			IF mcCartesianZMoveAbsolute.Done THEN
				bMissingCaps						:= TRUE;
				bCycleDone;
				mcCartesianZMoveAbsolute.Execute	:= FALSE;
				eRunningState						:= E_CapPreScrewer.eReady;	
			END_IF
			
		ELSE
			mcCartesianZMoveAbsolute.Execute		:= NOT stParameters.bVacuumDeactivate;		
			mcCartesianZMoveAbsolute.Position		:= stParameters.lrTopZPosition;
			mcCartesianZMoveAbsolute.Acceleration	:= SEL(GVL_Recipe.iCapSorterProductType = 0 ,stParameters.lrPickerAcceleration , 150.0);//stParameters.lrPickerAcceleration;
//			mcCartesianZMoveAbsolute.Acceleration	:= stParameters.lrPickerAcceleration;
			mcCartesianZMoveAbsolute.Deceleration	:= stParameters.lrPickerAcceleration;
			mcCartesianZMoveAbsolute.Velocity		:= stParameters.lrPickerSpeed;
			tonCapCatcher.IN						:= FALSE;
			
			IF mcCartesianZMoveAbsolute.Busy OR stParameters.bVacuumDeactivate THEN
				mcCartesianZMoveAbsolute.Execute		:= FALSE;
				eRunningState 							:= E_CapPreScrewer.eTransferingVertical; 
			END_IF
			
        
		END_IF		
			
			//przepisuje do rejestrów nakretki które kartezjan pobrał
			aCapPresence[1] := bCapSucker[1];
			aCapPresence[2] := bCapSucker[2];
			aCapPresence[3] := bCapSucker[3];
			aCapPresence[4] := bCapSucker[4];						

		
		
	(*Jazda w górę, zamknięcie łapek i załączenie jazdy w bok*)	
	E_CapPreScrewer.eTransferingVertical:
		
		IF NOT bCapSucker[1] OR NOT bCapSucker[2] OR NOT bCapSucker[3] OR NOT bCapSucker[4] THEN
            bCapBlow1						:= NOT bCapSucker[1];
            bCapBlow2						:= NOT bCapSucker[2];
            bCapBlow3						:= NOT bCapSucker[3];
            bCapBlow4						:= NOT bCapSucker[4];						
			bCapsBlowON						:= TRUE;
		END_IF
		
		//Kleją się kulki 
		IF NOT stParameters.bVacuumDeactivate THEN					
			IF CartesianZAxisRef.NcToPlc.ActPos > stParameters.lrPickZPosition + 10.0 THEN
				mcCartesianZMoveAbsolute2.Execute		:= NOT stParameters.bVacuumDeactivate;		
				mcCartesianZMoveAbsolute2.Position		:= stParameters.lrTopZPosition;
				mcCartesianZMoveAbsolute2.Acceleration	:= stParameters.lrPickerAcceleration;
				mcCartesianZMoveAbsolute2.Deceleration	:= stParameters.lrPickerAcceleration;
				mcCartesianZMoveAbsolute2.Velocity		:= stParameters.lrPickerSpeed;
			END_IF
		END_IF


		IF CartesianZAxisRef.NcToPlc.ActPos > stParameters.lrCapCatcherZPosition OR (CartesianZAxisRef.NcToPlc.ActPos > stParameters.lrTopZPosition - stParameters.lrBendingDistance) THEN
			bCapCatcher1							:= TRUE;
			bCapCatcher2							:= true;
			bCapCatcher3							:= true;
			bCapCatcher4							:= true;
			tonCapCatcher.IN						:= stParameters.bVacuumDeactivate;
		END_IF	
		
		mcCartesianZMoveAbsolute.Execute		:= tonCapCatcher.Q;	
		
		//Dodać sprawdzenie czy gotowy chwytak słomek !!!!!
		//Sprawdzenie pozycji osi pionowej Z i czy wysunięty siłownik chwytaka słomek
		IF ((CartesianZAxisRef.NcToPlc.ActPos > stParameters.lrTopZPosition - stParameters.lrBendingDistance) OR
			mcCartesianZMoveAbsolute.Done) AND (tonStrawCatcherOut.Q OR NOT stParameters.bStrawCatcherON) THEN
			//Jedź osią poziomą X na pozycję pick
				mcCartesianZMoveAbsolute2.Execute		:= FALSE;
				bCapsBlowON								:= FALSE;
				eRunningState 							:= E_CapPreScrewer.eTransferingHorizontal;
				tonCapCatcher.IN						:= FALSE;
		END_IF
	
	(*Przejazd w poziomie*)	
	E_CapPreScrewer.eTransferingHorizontal:	
	
			bCapCatcher1							:= TRUE;//bCapSucker1;
			bCapCatcher2							:= TRUE;//bCapSucker2;
			bCapCatcher3							:= TRUE;//bCapSucker3;
			bCapCatcher4							:= TRUE;//bCapSucker4;
	
		mcCartesianYMoveAbsolute.Position			:= stParameters.lrPlaceYPosition;
		mcCartesianYMoveAbsolute.Acceleration		:= stParameters.lrPickerAcceleration;
		mcCartesianYMoveAbsolute.Deceleration		:= stParameters.lrPickerAcceleration;
		mcCartesianYMoveAbsolute.Velocity			:= stParameters.lrPickerSpeed;
		mcCartesianYMoveAbsolute.Execute			:= TRUE;
		
		IF (CartesianYAxisRef.NcToPlc.ActPos > 200.0 (*stParameters.lrPlaceYPosition - stParameters.lrBendingDistance*)) OR
			mcCartesianYMoveAbsolute.Done AND NOT mcCartesianZMoveAbsolute.Execute THEN			

			//Podjedź robotem w dól	
			mcCartesianZMoveAbsolute.Execute			:= TRUE;		
			mcCartesianZMoveAbsolute.Position			:= stParameters.lrCartesianCatchZPosition;
			mcCartesianZMoveAbsolute.Acceleration		:= stParameters.lrPickerAcceleration;
			mcCartesianZMoveAbsolute.Deceleration		:= stParameters.lrPickerAcceleration;
			mcCartesianZMoveAbsolute.Velocity			:= stParameters.lrPickerSpeed;
		END_IF
		
		//Jak obie pozycje osiągnięte 
		IF mcCartesianZMoveAbsolute.Done THEN
			mcCartesianZMoveAbsolute.Execute		:= FALSE;
		END_IF
			
		//Jak ak obie pozycje osiągnięte to zamykamy chwytaki i następny krok
		IF stParameters.bStrawCatcherON AND CartesianYAxisRef.NcToPlc.ActPos >= stParameters.lrPlaceYPosition THEN
			//Zamknij chwytaki słomek
			bStrawCatchersOpen						:= FALSE;
			bStrawCatchersClose						:= TRUE;	
		END_IF
		
			
		IF  mcCartesianYMoveAbsolute.Done AND mcCartesianZMoveAbsolute.Done THEN
			//Reset komendy ruchu osi
			mcCartesianYMoveAbsolute.Execute		:= FALSE;
			mcCartesianZMoveAbsolute.Execute		:= FALSE;
			
				//Ustaw pozycję wirtualnej osi tak samo jak na osi Z
			fbVirtualAxis.fPosition						:= CartesianZAxisRef.NcToPlc.ActPos;
			fbVirtualAxis.SetPosAbsClearLag(bExecute	:= TRUE);
				
				IF fbVirtualAxis.pSetPos.Busy THEN
					//Następny krok
					eRunningState						:= E_CapPreScrewer.eVerticalDownToCatchPos;	
				END_IF
		END_IF		
		
	(*Przejazd w dól do pozycji chwytanija rurki*)		
	E_CapPreScrewer.eVerticalDownToCatchPos:
		fbVirtualAxis.SetPosAbsClearLag(bExecute				:= FALSE);
		
		//Jak ak obie pozycje osiągnięte to zamykamy chwytaki i następny krok
		IF stParameters.bStrawCatcherON THEN
			//Zamknij chwytaki słomek
			bStrawCatchersOpen						:= FALSE;
			bStrawCatchersClose						:= TRUE;	
		END_IF
				
		IF tonPlacePermission.Q AND ((bCapCatcher1 OR NOT bCapCatcher1) AND (bCapCatcher2  OR NOT bCapCatcher2) AND
									(bCapCatcher3  OR NOT bCapCatcher3) AND(bCapCatcher4  OR NOT bCapCatcher4)) AND (tonStrawCatcher1Close.Q OR NOT stParameters.bStrawCatcherON) THEN				
				bCapCatcher1						:= TRUE;
				bCapCatcher2						:= TRUE;
				bCapCatcher3						:= TRUE;
				bCapCatcher4						:= TRUE;						
				eRunningState						:= E_CapPreScrewer.eAxisGearIn;
		END_IF
		
			//Następny krok
			//IF stParameters.bStrawCatcherON THEN
			//	eRunningState						:= E_CapPreScrewer.eCatching;	
			//ELSE
			//	eRunningState						:= E_CapPreScrewer.ePlacing;	
			//END_IF				
		//END_IF
	
	
	E_CapPreScrewer.eAxisGearIn:
		fbGearInCatcherAxis.Enable						:= stParameters.bStrawCatcherON;
		fbGearInCatcherAxis.GearRatio					:= 1;
		fbGearInAxisZ.Enable							:= TRUE;
		fbGearInAxisZ.GearRatio							:= SEL(stParameters.bStrawCatcherON, 1.0, 0.0000000001);
		
		
			IF (fbGearInCatcherAxis.InGear OR NOT stParameters.bStrawCatcherON) AND fbGearInAxisZ.InGear AND (tonStrawCatcher1Close.Q (*AND tonStrawCatcher2Close.Q*)
					OR (bStrawCatcherOpen1 AND bStrawCatcherOpen2 AND bStrawCatcherOpen3 AND bStrawCatcherOpen4))  THEN
				IF stParameters.bStrawCatcherON THEN
					eRunningState						:= E_CapPreScrewer.eCatching;	
				ELSE
					eRunningState						:= E_CapPreScrewer.ePlacing;	
				END_IF					
			END_IF		

	
	//Sprawdzanie czy chwytaki zamknięte i opuszczenie chwytaków do dolnej pozycji
	E_CapPreScrewer.eCatching:
		fbVirtualAxis.fPosition							:= (stParameters.LrCheckStrawCatcherActuatorZPosition - stParameters.lrStrawInsertDistance);	//Pozycja sprawdzania cofnięcia krabów
		fbVirtualAxis.fVelocity							:= SEL(stParameters.lrCatcherSpeed > 1094.0, stParameters.lrCatcherSpeed, 1094.0 );       						
		bVirtualMove									:= TRUE;				
	
	IF (CatcherAxisRef.NcToPlc.ActPos + stParameters.lrCatcherHightSV) <= (stParameters.lrCartesianCatchZPosition - (stParameters.lrCapHight + 25.0)) THEN	//+25
		fbGearInAxisZ.GearRatio								:= 1;
	END_IF
	
	//IF (CatcherAxisRef.NcToPlc.ActPos + stParameters.lrCatcherHightSV) <= (stParameters.lrCartesianCatchZPosition-(stParameters.lrCapHight)) THEN
	//	fbGearInAxisZ.GearRatio							:= 1;
	//END_IF
	
			//Otwórz chwytaki słomek
		IF CartesianZAxisRef.NcToPlc.ActPos <= stParameters.lrStrawCatcherZPosition THEN					
			bStrawCatchersOpen							:= TRUE;
			bStrawCatchersClose							:= FALSE;
			
				IF tonStrawCatcher1Open.Q AND tonStrawCatcher2Open.Q AND tonStrawCatcher3Open.Q AND tonStrawCatcher4Open.Q THEN																				
					//Cofnij chwytaki słomek
					bStrawCatcherActuatorIn				:= TRUE;
					bStrawCatcherActuatorOut			:= FALSE;				
				END_IF	
			
		END_IF		
		
		
		// 10mm stały offset - wysokość nad butelką
		//IF (CatcherAxisRef.NcToPlc.ActPos <= 1.0) OR (CatcherAxisRef.NcToPlc.ActPos <= ((stParameters.lrBottleHight) - stParameters.lrCatcherHightSV-20.0)) THEN	//20
		IF (CatcherAxisRef.NcToPlc.ActPos <= 1.0) OR (CatcherAxisRef.NcToPlc.ActPos + 32 <= ((stParameters.lrBottleHight + 10.0) - stParameters.lrCatcherHightSV)) THEN		
			fbGearInCatcherAxis.GearRatio				:= 0.0000000001;
				
				IF bStrawCatcherIn THEN
					fbGearInCatcherAxis.GearRatio		:= 0.0000000001;
					bVirtualMove						:= FALSE;	
					bStepButton							:= FALSE;
					eRunningState						:= E_CapPreScrewer.ePlacing;
				END_IF		
			
		END_IF
	


	
	//Czekaj aż chwytak słomek dojedzie do dołu i zacznij ruch osi pionowej Z
	E_CapPreScrewer.ePlacing:		
		IF stParameters.lrScrewFinding > 0 THEN
			eRunningState								:= E_CapPreScrewer.eFinding;
		ELSE
			lrPreScrewerAxisSavedPosition				:= PreScrewerAxisRef.NcToPlc.ActPos;	//zapisywanie pozycji przed zakrecaniem		
			fbVirtualAxis.fPosition						:= SEL(stParameters.bStrawCatcherON, stParameters.lrPlaceZPosition, stParameters.lrPlaceZPosition - stParameters.lrStrawInsertDistance);
			fbVirtualAxis.fVelocity						:= SEL(stParameters.lrCatcherSpeed > 1094.0, stParameters.lrCatcherSpeed, 1094.0 );    
			bVirtualMove								:= TRUE;
			
			eRunningState								:= E_CapPreScrewer.ePreScrewing;
		END_IF
	
	E_CapPreScrewer.eFinding:
		fbVirtualAxis.fPosition							:= SEL(stParameters.bStrawCatcherON, stParameters.lrScrewerStartZPosition, stParameters.lrScrewerStartZPosition-stParameters.lrStrawInsertDistance);
		fbVirtualAxis.fVelocity							:= SEL(stParameters.lrCatcherSpeed > 1094.0, stParameters.lrCatcherSpeed, 1094.0 );
		fbVirtualAxis.fAcceleration						:= stParameters.lrCatcherAcceleration; 
		fbVirtualAxis.fDeceleration						:= stParameters.lrCatcherAcceleration; 
		fbVirtualAxis.fJerk								:= stParameters.lrCatcherJerk;        		
			                                            
		bVirtualMove									:= TRUE;
		                                                
			IF ABS(fbVirtualAxis.Axis.NcToPlc.ActPos - fbVirtualAxis.fPosition) <= 0.5 THEN 

             
				bCapSucker[1]								:= FALSE;
				bCapSucker[2]								:= FALSE;
				bCapSucker[3]								:= FALSE;
				bCapSucker[4]								:= FALSE;
    	                                                
				mcPreScrewerMoveRelative.Distance		:= stParameters.lrScrewFinding * -1.0;
				mcPreScrewerMoveRelative.Acceleration	:= stParameters.lrScrewAcceleration;
				mcPreScrewerMoveRelative.Deceleration	:= stParameters.lrScrewAcceleration;
				mcPreScrewerMoveRelative.Velocity		:= stParameters.lrScrewSpeed;
				mcPreScrewerMoveRelative.Execute		:= TRUE;
			END_IF
			
					IF mcPreScrewerMoveRelative.Done OR ABS(PreScrewerAxisRef.NcToPlc.PosDiff) > 60.0 OR mcPreScrewerMoveRelative.Error THEN
						bVirtualMove							:= FALSE;
						mcPreScrewerMoveRelative.Execute		:= FALSE;
						eRunningState							:= E_CapPreScrewer.eScrewing;
					END_IF	
	
	E_CapPreScrewer.ePreScrewing:

	IF fbVirtualAxis.Axis.Status.Moving THEN
		bVirtualMove											:= FALSE;
		eRunningState											:= E_CapPreScrewer.eScrewing;
	END_IF
	
	
	E_CapPreScrewer.eScrewing:
		
				//8mm przed zakręcaniem synchronizuję prędkościowo posuw kartezjana
			IF CartesianZAxisRef.NcToPlc.ActPos <= stParameters.lrScrewerStartZPosition + 20 THEN	//+8
				
				
				fbVirtualAxis.fPosition					:= SEL(stParameters.bStrawCatcherON, stParameters.lrPlaceZPosition, stParameters.lrPlaceZPosition - stParameters.lrStrawInsertDistance);
				fbVirtualAxis.fVelocity					:= stParameters.lrPickerSpeedWhenScrewer;   
				fbVirtualAxis.fAcceleration				:= 100_000_000.0;
				fbVirtualAxis.fDeceleration				:= 100_000_000.0;
				fbVirtualAxis.fJerk						:= 100_000_000;//100_000_000_000;       
				bVirtualMove							:= TRUE;
			
						//1.0mm przed pozycją zakręcania załączam obrót
					IF CartesianZAxisRef.NcToPlc.ActPos <= stParameters.lrScrewerStartZPosition + 2.5 OR stVirtualMove_Out.Done THEN	
						lrPreScrewerAxisSavedPosition			:= PreScrewerAxisRef.NcToPlc.ActPos;	//zapisywanie pozycji przed zakrecaniem	potrzebna dla opcji otwierania chwytaków butelek	
						bCapSucker[1]							:= FALSE;
						bCapSucker[2]							:= FALSE;
						bCapSucker[3]							:= FALSE;
						bCapSucker[4]							:= FALSE;
						mcPreScrewerMoveRelative.Execute		:= TRUE;
						mcPreScrewerMoveRelative.Distance		:= stParameters.lrScrewDistance;
						mcPreScrewerMoveRelative.Acceleration	:= stParameters.lrScrewAcceleration;
						mcPreScrewerMoveRelative.Deceleration	:= stParameters.lrScrewAcceleration;
						mcPreScrewerMoveRelative.Velocity		:= stParameters.lrScrewSpeed;	
						eRunningState							:= E_CapPreScrewer.eFinished;	
					END_IF	
			END_IF
	
	//Kończenie cyklu zakręcania - otwarcie chwytaka
	E_CapPreScrewer.eFinished:		
					//otwórz centrowniki butelek
		//IF (GVL_Recipe.bCapSorterPreScrewerCatchAngleOpenEnaShow AND
		//	ABS(PreScrewerAxisRef.NcToPlc.ActPos - lrPreScrewerAxisSavedPosition) >= GVL_Recipe.lrCapSorterPreScrewerCatchAngleOpenSV) THEN
		//	bBottleCatcherCatchTemp					:= FALSE;
		//END_IF
	
		IF PreScrewerAxisRef.NcToPlc.PosDiff > 100.0 OR (mcPreScrewerMoveRelative.Done AND (stVirtualMove_Out.Done OR stVirtualMove2_Out.Done)) THEN
//			bBottleCatcherCatchTemp							:= FALSE;
			bCapCatcher1									:= FALSE;
		 	bCapCatcher2									:= FALSE;
		 	bCapCatcher3									:= FALSE;
		 	bCapCatcher4									:= FALSE;
			mcPreScrewerMoveRelative.Execute				:= FALSE;
			bVirtualMove									:= FALSE;
			
				IF fbVirtualAxis.Axis.Status.Moving THEN
					fbVirtualAxis.Halt(bExecute := TRUE);
				ELSIF PreScrewerAxisRef.Status.Moving THEN
					mcPreScrewerStop.Execute	:= TRUE;					
				ELSE
					mcPreScrewerStop.Execute	:= FALSE;
					fbVirtualAxis.Halt(bExecute := FALSE);
					fbGearInCatcherAxis.Enable				:= FALSE;
					fbGearInAxisZ.Enable					:= FALSE;
					eRunningState							:= E_CapPreScrewer.eGearOut;
				END_IF	
		END_IF
		
	E_CapPreScrewer.eGearOut:
		fbGearOutAxisZ.Execute								:= TRUE;
		fbGearOutCatcherAxis.Execute						:= TRUE;
	
			IF NOT CartesianZAxisRef.Status.Coupled AND NOT CatcherAxisRef.Status.Coupled THEN
				fbGearOutAxisZ.Execute						:= FALSE;
				fbGearOutCatcherAxis.Execute				:= FALSE;
				eRunningState								:= E_CapPreScrewer.eReturning1;
			END_IF
	
	//Powrót na górną pozycję
	E_CapPreScrewer.eReturning1:
	
		tonWaitInPlacePos.IN						:= TRUE;
		mcPreScrewerStop.Execute					:= TRUE;
		bCapCatcher1								:= FALSE;
		bCapCatcher2								:= FALSE;
		bCapCatcher3								:= FALSE;
		bCapCatcher4								:= FALSE;
		
		
		IF tonWaitInPlacePos.Q AND NOT PreScrewerAxisRef.Status.Moving THEN
			

		
			tonWaitInPlacePos.IN					:= FALSE;
//			bBottleCatcherCatchTemp					:= FALSE;		
			mcPreScrewerStop.Execute				:= FALSE;
			mcCartesianZMoveAbsolute.Execute		:= TRUE;
			mcCartesianZMoveAbsolute.Position		:= stParameters.lrTopZPosition;
			mcCartesianZMoveAbsolute.Acceleration	:= SEL(GVL_Recipe.iCapSorterProductType = 0 ,stParameters.lrPickerAcceleration , 150.0);
//			mcCartesianZMoveAbsolute.Acceleration	:= stParameters.lrPickerAcceleration;
			mcCartesianZMoveAbsolute.Deceleration	:= stParameters.lrPickerAcceleration;
			mcCartesianZMoveAbsolute.Velocity		:= stParameters.lrPickerSpeed;
			
			IF mcCartesianZMoveAbsolute.Busy THEN
				bCapBlow1								:= TRUE;
        		bCapBlow2								:= TRUE;
        		bCapBlow3								:= TRUE;
        		bCapBlow4								:= TRUE;	

					IF CartesianZAxisRef.NcToPlc.ActPos >= stParameters.lrScrewerStartZPosition	THEN
						bCapsBlowON								:= TRUE;
						mcCartesianZMoveAbsolute.Execute		:= FALSE;
						eRunningState							:= E_CapPreScrewer.eReturning2;
					END_IF		                                   
			END_IF
			
		END_IF
		

		
	//Powrót po osi X	
	E_CapPreScrewer.eReturning2:
		bBottleCatcherCatchTemp					:= FALSE;

		
		
		IF CartesianZAxisRef.NcToPlc.ActPos > stParameters.lrScrewerStartZPosition + 15.0 THEN
			mcCartesianZMoveAbsolute2.Execute		:= TRUE;
			mcCartesianZMoveAbsolute2.Position		:= stParameters.lrTopZPosition;
			mcCartesianZMoveAbsolute2.Acceleration	:= stParameters.lrPickerAcceleration;
			mcCartesianZMoveAbsolute2.Deceleration	:= stParameters.lrPickerAcceleration;
			mcCartesianZMoveAbsolute2.Velocity		:= stParameters.lrPickerSpeed;			
		END_IF
	
		IF (CartesianZAxisRef.NcToPlc.ActPos > stParameters.lrTopZPosition - stParameters.lrBendingDistance) OR
			mcCartesianZMoveAbsolute.Done THEN
			mcCatcherMoveAbsolute.Execute			:= TRUE;		
			mcCatcherMoveAbsolute.Position			:= stParameters.lrCatcherCatchingPosition;
			mcCatcherMoveAbsolute.Acceleration		:= stParameters.lrCatcherAcceleration;
			mcCatcherMoveAbsolute.Deceleration		:= stParameters.lrCatcherAcceleration;
			mcCatcherMoveAbsolute.Velocity			:= stParameters.lrCatcherSpeed;

//SEL(P190_CapFeeder.stMover2Status.bInPlacePosition, GVL_Recipe.lrCapSorterPreScrewerPickXMover1PositionShow, GVL_Recipe.lrCapSorterPreScrewerPickXMover2PositionShow

			
			//Jedź osią poziomą X na pozycję pick
			mcCartesianYMoveAbsolute.Execute		:= TRUE;
			{warning 'Przerobić, dodać parametry obu pozycji wózków do struktury parametrów, FB_CapPreScrewer.Running --> 624'}
			mcCartesianYMoveAbsolute.Position		:= SEL(bMover1InPickPos, GVL_Recipe.lrCapSorterPreScrewerPickXMover1PositionShow, GVL_Recipe.lrCapSorterPreScrewerPickXMover2PositionShow);
			mcCartesianYMoveAbsolute.Acceleration	:= stParameters.lrPickerAcceleration;
			mcCartesianYMoveAbsolute.Deceleration	:= stParameters.lrPickerAcceleration;
			mcCartesianYMoveAbsolute.Velocity		:= stParameters.lrPickerSpeed;
			//Ustaw obracarkę do pozycji początkowej
			
			mcPreScrewerMoveRelative.Distance		:= -1 * DINT_TO_LREAL(LREAL_TO_DINT(PreScrewerAxisRef.NcToPlc.SetPos) MOD 360); 
			mcPreScrewerMoveRelative.Execute		:= mcPreScrewerMoveRelative.Distance<>0 AND NOT mcPreScrewerMoveRelative.Error;
			mcPreScrewerMoveRelative.Acceleration	:= stParameters.lrScrewAcceleration;
			mcPreScrewerMoveRelative.Deceleration	:= stParameters.lrScrewAcceleration;
			mcPreScrewerMoveRelative.Velocity		:= stParameters.lrScrewSpeed;
			
		END_IF
		IF CartesianZAxisRef.NcToPlc.ActPos > stParameters.lrPlaceZPosition + 20 THEN
			bPlaceDone								:= TRUE;
		END_IF
		IF (*bPlaceDone AND*) mcCartesianYMoveAbsolute.Done AND mcCartesianZMoveAbsolute2.Done AND
			 mcCatcherMoveAbsolute.Done AND NOT bCapBlow1 AND NOT bCapBlow2 AND NOT bCapBlow3 AND NOT bCapBlow4 THEN
				 IF mcPreScrewerMoveRelative.Distance=0 OR mcPreScrewerMoveRelative.Done THEN
					mcCartesianYMoveAbsolute.Execute		:= FALSE;
 					mcCartesianZMoveAbsolute.Execute		:= FALSE;
					mcCartesianZMoveAbsolute2.Execute		:= FALSE;
					mcCatcherMoveAbsolute.Execute			:= FALSE;
					mcPreScrewerMoveRelative.Execute		:= FALSE;
					eRunningState				:= E_CapPreScrewer.eDone;
				END_IF
		END_IF
		
		//Dodatkowy przedmuch ssawek
		(*IF (CartesianZAxisRef.NcToPlc.ActPos > (stParameters.lrPlaceZPosition + stParameters.lrHeightAdditionalBlow)) THEN
			bAdditionalBlow							S= NOT tonBlowOFF.IN;	
		
			IF NOT bAdditionalBlow THEN
				bCapsBlowON							R= tonBlowOFF.Q;
			END_IF

			bCapsBlowON								S= bAdditionalBlow;
			bCapBlow1 := bCapBlow2 := bCapBlow3 := bCapBlow4 := bAdditionalBlow;
		END_IF*)
			
	E_CapPreScrewer.eDone:
		mcPreScrewerStop.Execute				:= TRUE;
	
		IF mcPreScrewerStop.Done THEN
			mcPreScrewerStop.Execute			:= FALSE;
			bAdditionalBlow						:= FALSE;
			bCycleNotDone						:= FALSE;
			bCapsBlowON							:= FALSE;
			bPlaceDone							:= TRUE;
			bCycleDone							:= TRUE;
			eState								:= E_Station.eDone;
			eRunningState						:= E_CapPreScrewer.eReady;	
		END_IF	

	(*Cykl nie zakończony - przerwany - chyba nie potrzebny*)
	E_CapPreScrewer.eNotDone:
		bCapsBlowON							:= FALSE;
		eState								:= E_Station.eDone;
		eRunningState						:= E_CapPreScrewer.eReady;




END_CASE

tonCapCatcher(PT := T#60MS);
END_ACTION

ACTION RunningCam:

tonVacuumWatchdog(PT	:= stParameters.tTimeVacuumWatchdog);
bStopAllowed	:= eRunningState = E_CapPreScrewer.eReady OR eRunningState = E_CapPreScrewer.eVerticalDownToCatchPos;

//Otwieranie chwytaków
//bBottleCatcherCatchTemp		R= CartesianZAxisRef.NcToPlc.ActPos < stParameters.lrGripperOpenPosition;
GVL_VIS.bCapSorterPreScrewerBottleCatcherCatch	:= bBottleCatcherCatchTemp AND bCapSorterPreScrewerBottleCatcherEnableShow;
	
tonWaitInPlacePos(PT	:= stParameters.tWaitInPlacePos);
//tonWaitInPlacePos(PT 	:= T#200MS);
eLastRunningState	:= eRunningState;

CASE eRunningState OF

//====================================
	
	(*Oczekiwanie na wykonanie pojedynczego cyklu*)
	E_CapPreScrewer.eReady:

		
		IF NOT bCycleDone AND NOT bCycleNotDone THEN  
                                      	
			IF bRun THEN 
				fbVirtualAxis.fAcceleration				:= stParameters.lrPickerAcceleration;	//100_000_000.0;
				fbVirtualAxis.fDeceleration				:= stParameters.lrPickerAcceleration;	//100_000_000.0;
				fbVirtualAxis.fJerk						:= stParameters.lrPickerJerk;// 	1_000_000;//100_000_000_000;  

				iRejectCase					:= 0;
				bRejectDone					:= FALSE;
				bReject						:= FALSE;
				bTubeReject					:= FALSE;
				
				//Przygotuj do cyklu - otwórz chwytaki
				bCapCatcher1				:= FALSE;
				bCapCatcher2				:= FALSE;
				bCapCatcher3				:= FALSE;
				bCapCatcher4				:= FALSE;
	
				//Wyłącz ssawki
				bCapSucker[1]				:= FALSE;
				bCapSucker[2]				:= FALSE;
				bCapSucker[3]				:= FALSE;
				bCapSucker[4]				:= FALSE;
				//Wyłącz odmuchy
				bCapBlower1					:= FALSE;
				bCapBlower2					:= FALSE;
				bCapBlower3					:= FALSE;
				bCapBlower4					:= FALSE;
				bCapsBlowON					:= FALSE;
				//Otwórz chwytaki słomek
				bStrawCatchersOpen			:= TRUE;
				bStrawCatchersClose			:= FALSE;
				//Cofnij chwytaki słomek
				bStrawCatcherActuatorIn		:= TRUE;
				bStrawCatcherActuatorOut	:= FALSE;
				//Podjedź robotem i chwytakiem słomek w górę jak cofnięty chwytak słomek
				IF tonStrawCatcherIn.Q THEN	
										
					mcCartesianZMoveAbsolute.Execute		:= TRUE;		
					mcCartesianZMoveAbsolute.Position		:= stParameters.lrTopZPosition;
					mcCartesianZMoveAbsolute.Acceleration	:= stParameters.lrPickerAcceleration;
					mcCartesianZMoveAbsolute.Deceleration	:= stParameters.lrPickerAcceleration;
					mcCartesianZMoveAbsolute.Velocity		:= stParameters.lrPickerSpeed;
					
					mcCatcherMoveAbsolute.Execute			:= TRUE;		
					mcCatcherMoveAbsolute.Position			:= stParameters.lrCatcherCatchingPosition;
					mcCatcherMoveAbsolute.Acceleration		:= stParameters.lrCatcherAcceleration;
					mcCatcherMoveAbsolute.Deceleration		:= stParameters.lrCatcherAcceleration;
					mcCatcherMoveAbsolute.Velocity			:= stParameters.lrCatcherSpeed;
					
					//Następny krok
					eRunningState						:= E_CapPreScrewer.ePreparingToPick;
					bCycleNotDone						:= TRUE;
					
				END_IF
				//Reset komendy ruchu osi X
				mcCartesianYMoveAbsolute.Execute		:= FALSE;
				
			END_IF
		END_IF
			
	(*Czekam na pozycję Z w górze i ruszam osią poziomą X na pozycję pobierania i czekam na obie pozycje*)
	E_CapPreScrewer.ePreparingToPick:
		IF (CartesianZAxisRef.NcToPlc.ActPos > stParameters.lrTopZPosition - stParameters.lrBendingDistance) OR
			mcCartesianZMoveAbsolute.Done THEN
			//Jedź osią poziomą X na pozycję pick
			mcCartesianYMoveAbsolute.Execute		:= TRUE;
			mcCartesianYMoveAbsolute.Position		:= stParameters.lrPickYPosition;
			mcCartesianYMoveAbsolute.Acceleration	:= stParameters.lrPickerAcceleration;
			mcCartesianYMoveAbsolute.Deceleration	:= stParameters.lrPickerAcceleration;
			mcCartesianYMoveAbsolute.Velocity		:= stParameters.lrPickerSpeed;
			//Nakrętka pobrana z wózka nr.1
			bMover1InPickPos						:= SEL((stParameters.lrPickYPosition-GVL_Recipe.lrCapSorterPreScrewerPickXMover1PositionShow) <= 0.5, FALSE, TRUE);
			
			//Ustaw obracarkę w pozycji
			mcPreScrewerMoveRelative.Distance		:=  -1 * DINT_TO_LREAL((LREAL_TO_DINT(PreScrewerAxisRef.NcToPlc.SetPos)+diPreSCrewerHomePos) MOD 360);
			mcPreScrewerMoveRelative.Execute		:= mcPreScrewerMoveRelative.Distance<>0;
			mcPreScrewerMoveRelative.Acceleration	:= stParameters.lrScrewAcceleration;
			mcPreScrewerMoveRelative.Deceleration	:= stParameters.lrScrewAcceleration;
			mcPreScrewerMoveRelative.Velocity		:= stParameters.lrScrewSpeed;
		END_IF
		//Jak obie pozycje osiągnięte to wysuń chwytak słomek i następny krok
		IF mcCartesianYMoveAbsolute.Done AND mcCartesianZMoveAbsolute.Done AND mcCatcherMoveAbsolute.Done THEN
			IF mcPreScrewerMoveRelative.Done OR mcPreScrewerMoveRelative.Distance =0 THEN
				//Reset komendy ruchu osi
				mcCartesianYMoveAbsolute.Execute		:= FALSE;
				mcCartesianZMoveAbsolute.Execute		:= FALSE;
				mcPreScrewerMoveRelative.Execute		:= FALSE;
				mcCatcherMoveAbsolute.Execute			:= FALSE;
				//Wysuń chwytaki słomek jesli to potrzebuje recepta        
				bStrawCatcherActuatorIn					:= NOT stParameters.bStrawCatcherON;
				bStrawCatcherActuatorOut				:= stParameters.bStrawCatcherON;    
				//Następny krok
				eRunningState							:= E_CapPreScrewer.ePicking;
			END_IF
		END_IF
		
	
	(*Zjeżdzam na osią pionową Z na pozycję chwytania i załączam ssawki*)		
	E_CapPreScrewer.ePicking:
		//Podjedź robotem w górę	
		mcCartesianZMoveAbsolute.Execute			:= TRUE;		
		mcCartesianZMoveAbsolute.Position			:= stParameters.lrPickZPosition;
		mcCartesianZMoveAbsolute.Acceleration		:= stParameters.lrPickerAcceleration;
		mcCartesianZMoveAbsolute.Deceleration		:= stParameters.lrPickerAcceleration;
		mcCartesianZMoveAbsolute.Velocity			:= stParameters.lrPickerSpeed;
		//Czekam na wykonanie ruchu
		IF mcCartesianZMoveAbsolute.Done THEN
			//Reset komendy ruchu osi
			mcCartesianZMoveAbsolute.Execute		:= FALSE;
			
			//Zeruje rejestry oraz załączanie ssawek
			 FOR i:=1 TO 4 DO
				 bCapSucker[i]						:= stParameters.bPickerActiv[i]; 
				 aCapPresence[i] 					:= FALSE;
			 END_FOR
	
			//Następny krok
			eRunningState							:= E_CapPreScrewer.eVacumCheckPart1;
		END_IF
	
	(*Sprawdzam czy zassane i jazda w górę*)	
	E_CapPreScrewer.eVacumCheckPart1:
		
		tonVacuumWatchdog.IN						:= TRUE;
		
		IF tonSuckedOk[1].Q = stParameters.bPickerActiv[1] AND tonSuckedOk[2].Q = stParameters.bPickerActiv[2]
			AND tonSuckedOk[3].Q = stParameters.bPickerActiv[3] AND tonSuckedOk[4].Q = stParameters.bPickerActiv[4] THEN
			tonVacuumWatchdog.IN					:= FALSE;
		
				FOR i:=1 TO 4 DO
					IF stParameters.bPickerActiv[i] AND stParameters.bStrawCatcherON AND NOT stMoverStatus.stSlotStatus[i].bTubePresent THEN
						bReject								:= TRUE;
						bTubeReject							:= TRUE;
						lrAxisZ_RejectOffset				:= 0.0;
					END_IF

					IF bMover1InPlacePos THEN
						diMover1VacuumRetry[i]		:= 0;
					ELSE
						diMover2VacuumRetry[i]		:= 0;
					END_IF	
				END_FOR 
				
			eRunningState 							:= E_CapPreScrewer.eVacumCheckPart2;
	
		ELSIF tonVacuumWatchdog.Q THEN
		
			FOR i:=1 TO 4 DO
				bCapSucker[i]							:= tonSuckedOk[i].Q;
				
				//robimy odrzut jeżeli zostanie wykryto brak słomki
				IF stParameters.bPickerActiv[i] AND stParameters.bStrawCatcherON AND NOT stMoverStatus.stSlotStatus[i].bTubePresent THEN
					bReject								:= TRUE;
					bTubeReject							:= TRUE;
					lrAxisZ_RejectOffset				:= 0.0;
				END_IF
				
						//Detekcja niepobranej nasadki --> odrzut aktywowany opcjonalnie z receptury
					IF stParameters.bPickerActiv[i] AND NOT tonSuckedOk[i].Q AND NOT stParameters.bVacuumDeactivate THEN
						bReject							:= SEL(stParameters.bRejectON, bReject, TRUE);
						lrAxisZ_RejectOffset			:= SEL(stParameters.bRejectON, lrAxisZ_RejectOffset, 13.0);	//offset dodatkowego zjazdu kartezjanem 
						
						IF bMover1InPlacePos THEN
							diMover1VacuumRetry[i]		:= diMover1VacuumRetry[i] + 1;
						ELSE	
							diMover2VacuumRetry[i]		:= diMover2VacuumRetry[i] + 1;
						END_IF
					ELSIF tonSuckedOk[i].Q OR stParameters.bVacuumDeactivate THEN
						IF 	bMover1InPlacePos THEN
							diMover1VacuumRetry[i]		:= 0;
						ELSE
							diMover2VacuumRetry[i]		:= 0;
						END_IF	
					END_IF	
	    	
			END_FOR
				tonVacuumWatchdog.IN					:= FALSE;
				eRunningState 							:= E_CapPreScrewer.eVacumCheckPart2;
	
		END_IF
		
		
	E_CapPreScrewer.eVacumCheckPart2:	
			
		//Jezeli nie jest przyssana zadna nasadka to pdjezdzamy na poz. ready oraz wystawiamy flage bMissingCaps
		IF bReject THEN
			Reject();
				IF bRejectDone THEN				
					eRunningState						:= E_CapPreScrewer.eReady;	
				END_IF		
		ELSIF NOT tonSuckedOk[1].Q AND NOT tonSuckedOk[2].Q AND NOT tonSuckedOk[3].Q AND NOT tonSuckedOk[4].Q THEN
			bCapSucker[1]							:= FALSE;
			bCapSucker[2]							:= False;
			bCapSucker[3]							:= False;
		    bCapSucker[4]							:= False;	
			mcCartesianZMoveAbsolute.Execute		:= TRUE;		
			mcCartesianZMoveAbsolute.Position		:= stParameters.lrTopZPosition;
			mcCartesianZMoveAbsolute.Acceleration	:= stParameters.lrPickerAcceleration;
			mcCartesianZMoveAbsolute.Deceleration	:= stParameters.lrPickerAcceleration;
			mcCartesianZMoveAbsolute.Velocity		:= stParameters.lrPickerSpeed;
			
			IF mcCartesianZMoveAbsolute.Done THEN
				bMissingCaps						:= TRUE;
				bCycleDone;
				mcCartesianZMoveAbsolute.Execute	:= FALSE;
				eRunningState						:= E_CapPreScrewer.eReady;	
			END_IF
			
		ELSE
			mcCartesianZMoveAbsolute.Execute		:= NOT stParameters.bVacuumDeactivate;		
			mcCartesianZMoveAbsolute.Position		:= stParameters.lrTopZPosition;
			mcCartesianZMoveAbsolute.Acceleration	:= SEL(GVL_Recipe.iCapSorterProductType = 0 ,stParameters.lrPickerAcceleration , 150.0);//stParameters.lrPickerAcceleration;
//			mcCartesianZMoveAbsolute.Acceleration	:= stParameters.lrPickerAcceleration;
			mcCartesianZMoveAbsolute.Deceleration	:= stParameters.lrPickerAcceleration;
			mcCartesianZMoveAbsolute.Velocity		:= stParameters.lrPickerSpeed;
			tonCapCatcher.IN						:= FALSE;
			
			IF mcCartesianZMoveAbsolute.Busy OR stParameters.bVacuumDeactivate THEN
				mcCartesianZMoveAbsolute.Execute		:= FALSE;
				eRunningState 							:= E_CapPreScrewer.eTransferingVertical; 
			END_IF
			
        
		END_IF		
			
			//przepisuje do rejestrów nakretki które kartezjan pobrał
			aCapPresence[1] := bCapSucker[1];
			aCapPresence[2] := bCapSucker[2];
			aCapPresence[3] := bCapSucker[3];
			aCapPresence[4] := bCapSucker[4];						

		
		
	(*Jazda w górę, zamknięcie łapek i załączenie jazdy w bok*)	
	E_CapPreScrewer.eTransferingVertical:
		
		IF NOT bCapSucker[1] OR NOT bCapSucker[2] OR NOT bCapSucker[3] OR NOT bCapSucker[4] THEN
            bCapBlow1						:= NOT bCapSucker[1];
            bCapBlow2						:= NOT bCapSucker[2];
            bCapBlow3						:= NOT bCapSucker[3];
            bCapBlow4						:= NOT bCapSucker[4];						
			bCapsBlowON						:= TRUE;
		END_IF
		
		//Kleją się kulki 
		IF NOT stParameters.bVacuumDeactivate THEN					
			IF CartesianZAxisRef.NcToPlc.ActPos > stParameters.lrPickZPosition + 10.0 THEN
				mcCartesianZMoveAbsolute2.Execute		:= NOT stParameters.bVacuumDeactivate;		
				mcCartesianZMoveAbsolute2.Position		:= SEL(stParameters.lrCartesianCatchZPosition > stParameters.lrTopZPosition, stParameters.lrTopZPosition, stParameters.lrCartesianCatchZPosition);
				mcCartesianZMoveAbsolute2.Acceleration	:= stParameters.lrPickerAcceleration;
				mcCartesianZMoveAbsolute2.Deceleration	:= stParameters.lrPickerAcceleration;
				mcCartesianZMoveAbsolute2.Velocity		:= stParameters.lrPickerSpeed;
			END_IF
		END_IF


		IF CartesianZAxisRef.NcToPlc.ActPos > stParameters.lrCapCatcherZPosition  THEN //OR (CartesianZAxisRef.Status.Moving)
			bCapCatcher1							:= TRUE;
			bCapCatcher2							:= true;
			bCapCatcher3							:= true;
			bCapCatcher4							:= true;
			tonCapCatcher.IN						:= stParameters.bVacuumDeactivate;
		END_IF	
		
		mcCartesianZMoveAbsolute.Execute		:= tonCapCatcher.Q;	
		
		//Dodać sprawdzenie czy gotowy chwytak słomek !!!!!
		//Sprawdzenie pozycji osi pionowej Z i czy wysunięty siłownik chwytaka słomek
		IF ((CartesianZAxisRef.NcToPlc.ActPos > stParameters.lrTopZPosition - stParameters.lrBendingDistance) OR
			mcCartesianZMoveAbsolute.Done) AND (tonStrawCatcherOut.Q OR NOT stParameters.bStrawCatcherON) THEN
			//Jedź osią poziomą X na pozycję pick
				mcCartesianZMoveAbsolute2.Execute		:= FALSE;
				bCapsBlowON								:= FALSE;
				eRunningState 							:= E_CapPreScrewer.eTransferingHorizontal;
				tonCapCatcher.IN						:= FALSE;
		END_IF
	
	(*Przejazd w poziomie*)	
	E_CapPreScrewer.eTransferingHorizontal:	
	
			bCapCatcher1							:= TRUE;//bCapSucker1;
			bCapCatcher2							:= TRUE;//bCapSucker2;
			bCapCatcher3							:= TRUE;//bCapSucker3;
			bCapCatcher4							:= TRUE;//bCapSucker4;
	
		mcCartesianYMoveAbsolute.Position			:= stParameters.lrPlaceYPosition;
		mcCartesianYMoveAbsolute.Acceleration		:= stParameters.lrPickerAcceleration;
		mcCartesianYMoveAbsolute.Deceleration		:= stParameters.lrPickerAcceleration;
		mcCartesianYMoveAbsolute.Velocity			:= stParameters.lrPickerSpeed;
		mcCartesianYMoveAbsolute.Execute			:= TRUE;
		
		IF (CartesianYAxisRef.NcToPlc.ActPos > 200.0 (*stParameters.lrPlaceYPosition - stParameters.lrBendingDistance*)) OR
			mcCartesianYMoveAbsolute.Done AND NOT mcCartesianZMoveAbsolute.Execute THEN			

			//Podjedź robotem w dól	
			mcCartesianZMoveAbsolute.Execute			:= TRUE;		
			mcCartesianZMoveAbsolute.Position			:= stParameters.lrCartesianCatchZPosition;
			mcCartesianZMoveAbsolute.Acceleration		:= stParameters.lrPickerAcceleration;
			mcCartesianZMoveAbsolute.Deceleration		:= stParameters.lrPickerAcceleration;
			mcCartesianZMoveAbsolute.Velocity			:= stParameters.lrPickerSpeed;
		END_IF
		
		//Jak obie pozycje osiągnięte 
		IF mcCartesianZMoveAbsolute.Done THEN
			mcCartesianZMoveAbsolute.Execute		:= FALSE;
		END_IF
			
		//Jak ak obie pozycje osiągnięte to zamykamy chwytaki i następny krok
		IF stParameters.bStrawCatcherON AND CartesianYAxisRef.NcToPlc.ActPos >= stParameters.lrPlaceYPosition THEN
			//Zamknij chwytaki słomek
			bStrawCatchersOpen						:= FALSE;
			bStrawCatchersClose						:= TRUE;	
		END_IF
		
			
		IF  mcCartesianYMoveAbsolute.Done AND mcCartesianZMoveAbsolute.Done THEN			
				//Ustaw pozycję wirtualnej osi tak samo jak na osi Z
			fbVirtualAxis.fPosition						:=  CartesianZAxisRef.NcToPlc.ActPos;
			fbVirtualAxis.SetPosAbsClearLag(bExecute	:= TRUE);
				
				IF fbVirtualAxis.pSetPos.Busy THEN
						//Reset komendy ruchu osi
					mcCartesianYMoveAbsolute.Execute	:= FALSE;
					mcCartesianZMoveAbsolute.Execute	:= FALSE;
					//Następny krok
					eRunningState						:= E_CapPreScrewer.eVerticalDownToCatchPos;	
				END_IF
		END_IF		
		
	(*Przejazd w dól do pozycji chwytanija rurki*)		
	E_CapPreScrewer.eVerticalDownToCatchPos:
		fbVirtualAxis.SetPosAbsClearLag(bExecute				:= FALSE);
		
		//Jak ak obie pozycje osiągnięte to zamykamy chwytaki i następny krok
		IF stParameters.bStrawCatcherON THEN
			//Zamknij chwytaki słomek
			bStrawCatchersOpen					:= FALSE;
			bStrawCatchersClose					:= TRUE;	
			//Generowanie krzywki
			CamCalculation();
			fbCamTableSelectCatcher.Execute		:= TRUE;	
			fbCamTableSelectAxisZ.Execute		:= TRUE;
		END_IF
				
			IF tonPlacePermission.Q AND (NOT stParameters.bStrawCatcherON OR (tonStrawCatcher1Close.Q AND fbCamTableSelectCatcher.Done AND fbCamTableSelectAxisZ.Done)) THEN	
					fbCamTableSelectCatcher.Execute		:= FALSE;
				   	fbCamTableSelectAxisZ.Execute		:= FALSE;
					bCapCatcher1						:= TRUE;
					bCapCatcher2						:= TRUE;
					bCapCatcher3						:= TRUE;
					bCapCatcher4						:= TRUE;						
					eRunningState						:= E_CapPreScrewer.eAxisGearIn;
			END_IF
		
	
	E_CapPreScrewer.eAxisGearIn:
	
		IF stParameters.bStrawCatcherON THEN
			fbCamInAxisZ.Execute						:= TRUE;
			fbCamInAxisCatcher.Execute					:= TRUE;
			
				IF fbCamInAxisZ.InSync AND fbCamInAxisCatcher.InSync THEN
					fbCamInAxisZ.Execute				:= FALSE;
					fbCamInAxisCatcher.Execute			:= FALSE;
				
				
					eRunningState					:= E_CapPreScrewer.ePositionOverBottle;	
					fbVirtualAxis.fPosition			:= (stParameters.LrCheckStrawCatcherActuatorZPosition - arrTableAxisZ[1,0]);	
					fbVirtualAxis.fVelocity			:= SEL(stParameters.lrCatcherSpeed > 1094.0, stParameters.lrCatcherSpeed, 1094.0 ); 
					bVirtualMove					:= TRUE;	
					eRunningState					:= E_CapPreScrewer.ePositionOverBottle;	
				END_IF	
		ELSE                            
			mcCartesianZMoveAbsolute.Execute		:= TRUE;		
			mcCartesianZMoveAbsolute.Position		:= stParameters.lrScrewerStartZPosition;
			mcCartesianZMoveAbsolute.Acceleration	:= stParameters.lrPickerAcceleration;
			mcCartesianZMoveAbsolute.Deceleration	:= stParameters.lrPickerAcceleration;
			mcCartesianZMoveAbsolute.Velocity		:= stParameters.lrPickerSpeed;
			eRunningState							:= E_CapPreScrewer.ePlacing;	
		END_IF	

	
	
	E_CapPreScrewer.ePositionOverBottle:		      			
		IF fbVirtualAxis.Axis.Status.Moving THEN
			bVirtualMove							:= FALSE;
			eRunningState							:= E_CapPreScrewer.eCatching;	
		END_IF
	
	
	//Sprawdzanie czy chwytaki zamknięte i opuszczenie chwytaków do dolnej pozycji
	E_CapPreScrewer.eCatching:
	
			//Otwórz chwytaki słomek
		IF CartesianZAxisRef.NcToPlc.ActPos <= stParameters.lrStrawCatcherZPosition THEN		
			bStrawCatchersOpen							:= TRUE;
			bStrawCatchersClose							:= FALSE;
			
				IF tonStrawCatcher1Open.Q AND tonStrawCatcher2Open.Q AND tonStrawCatcher3Open.Q AND tonStrawCatcher4Open.Q THEN																				
					//Cofnij chwytaki słomek
					bStrawCatcherActuatorIn				:= TRUE;
					bStrawCatcherActuatorOut			:= FALSE;				
				END_IF	
		END_IF		
						
				IF bStrawCatcherIn THEN	
					eRunningState						:= E_CapPreScrewer.ePlacing;
					fbVirtualAxis.fPosition				:= stParameters.lrScrewerStartZPosition - arrTableAxisZ[1,0];
					fbVirtualAxis.fVelocity				:= SEL(stParameters.lrCatcherSpeed > 1094.0, stParameters.lrCatcherSpeed, 1094.0 );    
					bVirtualMove						:= TRUE;
				END_IF		
			
		//END_IF
	


	
	//Czekaj aż chwytak słomek dojedzie do dołu i zacznij ruch osi pionowej Z
	E_CapPreScrewer.ePlacing:		
	
		IF stParameters.lrScrewFinding > 0 THEN
			eRunningState								:= E_CapPreScrewer.eFinding;
		ELSE
			eRunningState								:= E_CapPreScrewer.ePreScrewing;
		END_IF
	
	E_CapPreScrewer.eFinding:		                                                
			IF stParameters.bStrawCatcherON THEN
				IF ABS(fbVirtualAxis.Axis.NcToPlc.ActPos - fbVirtualAxis.fPosition) <= 3.0 THEN              
					bCapSucker[1]								:= FALSE;
					bCapSucker[2]								:= FALSE;
					bCapSucker[3]								:= FALSE;
					bCapSucker[4]								:= FALSE;
    	        	                                        
					mcPreScrewerMoveRelative.Distance		:= stParameters.lrScrewFinding * -1.0;
					mcPreScrewerMoveRelative.Acceleration	:= stParameters.lrScrewAcceleration;
					mcPreScrewerMoveRelative.Deceleration	:= stParameters.lrScrewAcceleration;
					mcPreScrewerMoveRelative.Velocity		:= stParameters.lrScrewSpeed;
					mcPreScrewerMoveRelative.Execute		:= TRUE;
				END_IF	
			ELSE	
				IF ABS(CartesianZAxisRef.NcToPlc.ActPos - mcCartesianZMoveAbsolute.Position) <= 3.0 THEN 
					bCapSucker[1]								:= FALSE;
					bCapSucker[2]								:= FALSE;
					bCapSucker[3]								:= FALSE;
					bCapSucker[4]								:= FALSE;
    	        	                                        
					mcPreScrewerMoveRelative.Distance		:= stParameters.lrScrewFinding * -1.0;
					mcPreScrewerMoveRelative.Acceleration	:= stParameters.lrScrewAcceleration;
					mcPreScrewerMoveRelative.Deceleration	:= stParameters.lrScrewAcceleration;
					mcPreScrewerMoveRelative.Velocity		:= stParameters.lrScrewSpeed;
					mcPreScrewerMoveRelative.Execute		:= TRUE;
				END_IF
			END_IF
			
					IF mcPreScrewerMoveRelative.Done OR ABS(PreScrewerAxisRef.NcToPlc.PosDiff) > 60.0 OR mcPreScrewerMoveRelative.Error THEN
						bVirtualMove							:= FALSE;
						mcPreScrewerMoveRelative.Execute		:= FALSE;
						eRunningState							:= E_CapPreScrewer.ePreScrewing;
					END_IF	
	
	E_CapPreScrewer.ePreScrewing:

		IF stParameters.bStrawCatcherON THEN
			IF ABS(fbVirtualAxis.Axis.NcToPlc.ActPos - fbVirtualAxis.fPosition)<=0.1 THEN
				bVirtualMove											:= FALSE;
				
				IF NOT	CartesianZAxisRef.Status.SynchronizedMotion AND NOT CartesianZAxisRef.Status.Moving THEN
					eRunningState				:= E_CapPreScrewer.eScrewing;
					mcCartesianZStop.Execute	:= FALSE;
					fbCamOutAxisZ.Execute		:= FALSE;
				ELSE
					fbCamOutAxisZ.Execute		:= TRUE;
					mcCartesianZStop.Execute	:= CartesianZAxisRef.Status.Moving;
				END_IF	
			END_IF
		ELSE
			IF mcCartesianZMoveAbsolute.Done THEN
				eRunningState						:= E_CapPreScrewer.eScrewing;
				mcCartesianZMoveAbsolute.Execute	:= FALSE;
			END_IF	
		END_IF
		
	
	
	E_CapPreScrewer.eScrewing:
	
			fbGearInAxisZ_Screwer.Execute			:= NOT CartesianZAxisRef.Status.Coupled AND NOT mcCartesianZStop.Busy;
			fbGearInAxisZ_Screwer.RatioNumerator 	:= (GVL_Recipe.lrCapSorterPreScrewerThreadPitchShow	* GVL_Recipe.lrCapSorterPreScrewerMultipleStartThreadShow * (-1));
			fbGearInAxisZ_Screwer.RatioDenominator	:= 360;
		
			IF CartesianZAxisRef.Status.Coupled THEN
						mcPreScrewerMoveRelative.Execute		:= TRUE;
						mcPreScrewerMoveRelative.Distance		:= stParameters.lrScrewDistance;
						mcPreScrewerMoveRelative.Acceleration	:= stParameters.lrScrewAcceleration;
						mcPreScrewerMoveRelative.Deceleration	:= stParameters.lrScrewAcceleration;
						mcPreScrewerMoveRelative.Velocity		:= stParameters.lrScrewSpeed;	
						eRunningState							:= E_CapPreScrewer.eFinished;	
			END_IF
	
	//Kończenie cyklu zakręcania - otwarcie chwytaka
	E_CapPreScrewer.eFinished:		
	
		IF PreScrewerAxisRef.NcToPlc.PosDiff > 100.0 OR mcPreScrewerMoveRelative.Done THEN
//			bBottleCatcherCatchTemp							:= FALSE;	
			bCapCatcher1									:= FALSE;
		 	bCapCatcher2									:= FALSE;
		 	bCapCatcher3									:= FALSE;
		 	bCapCatcher4									:= FALSE;
			mcPreScrewerMoveRelative.Execute				:= FALSE;
			bVirtualMove									:= FALSE;
			bCapBlow1										:= stParameters.bPickerActiv[1];
            bCapBlow2										:= stParameters.bPickerActiv[2];
            bCapBlow3										:= stParameters.bPickerActiv[3];
            bCapBlow4										:= stParameters.bPickerActiv[4];
			bCapSucker[1]									:= FALSE;
			bCapSucker[2]									:= FALSE;
			bCapSucker[3]									:= FALSE;
			bCapSucker[4]									:= FALSE;								
			
				IF PreScrewerAxisRef.Status.Moving THEN
					mcPreScrewerStop.Execute				:=	 TRUE;					
				ELSE
					lrAxisZSavedPosition					:= CartesianZAxisRef.NcToPlc.ActPos;
					mcPreScrewerStop.Execute				:= FALSE;
					fbGearInCatcherAxis.Enable				:= FALSE;
					eRunningState							:= E_CapPreScrewer.eGearOut;
				END_IF	
		END_IF
		
	E_CapPreScrewer.eGearOut:
		fbGearOutAxisZ.Execute								:= TRUE;
		fbCamOutAxisCatcher.Execute							:= TRUE;
	
			IF NOT CartesianZAxisRef.Status.Coupled AND NOT CatcherAxisRef.Status.SynchronizedMotion THEN
				fbGearOutAxisZ.Execute						:= FALSE;
				fbCamOutAxisCatcher.Execute					:= FALSE;
				eRunningState								:= E_CapPreScrewer.eReturning1;
			END_IF
	
	//Powrót na górną pozycję
	E_CapPreScrewer.eReturning1:
	
		tonWaitInPlacePos.IN						:= TRUE;
		mcPreScrewerStop.Execute					:= TRUE;		

		IF tonWaitInPlacePos.Q THEN
			

		
			tonWaitInPlacePos.IN					:= FALSE;
//			bBottleCatcherCatchTemp					:= FALSE;		
			mcPreScrewerStop.Execute				:= FALSE;
			mcCartesianZMoveAbsolute.Execute		:= TRUE;
			mcCartesianZMoveAbsolute.Position		:= stParameters.lrTopZPosition;
			mcCartesianZMoveAbsolute.Acceleration	:= SEL(GVL_Recipe.iCapSorterProductType = 0 ,stParameters.lrPickerAcceleration , 150.0);
//			mcCartesianZMoveAbsolute.Acceleration	:= stParameters.lrPickerAcceleration;
			mcCartesianZMoveAbsolute.Deceleration	:= stParameters.lrPickerAcceleration;
			mcCartesianZMoveAbsolute.Velocity		:= stParameters.lrPickerSpeed;
			
			IF mcCartesianZMoveAbsolute.Busy THEN
				mcCartesianZMoveAbsolute.Execute		:= FALSE;
				eRunningState							:= E_CapPreScrewer.eReturning2;
			END_IF
			
		END_IF

		
	//Powrót po osi X	
	E_CapPreScrewer.eReturning2:
		bBottleCatcherCatchTemp					:= FALSE;
		bCapsBlowON								:= CartesianZAxisRef.NcToPlc.ActPos > lrAxisZSavedPosition + 10.0;
		
		IF CartesianZAxisRef.NcToPlc.ActPos > stParameters.lrScrewerStartZPosition + 15.0 THEN
			mcCartesianZMoveAbsolute2.Execute		:= TRUE;
			mcCartesianZMoveAbsolute2.Position		:= stParameters.lrTopZPosition;
			mcCartesianZMoveAbsolute2.Acceleration	:= stParameters.lrPickerAcceleration;
			mcCartesianZMoveAbsolute2.Deceleration	:= stParameters.lrPickerAcceleration;
			mcCartesianZMoveAbsolute2.Velocity		:= stParameters.lrPickerSpeed;			
		END_IF
	
		IF (CartesianZAxisRef.NcToPlc.ActPos > stParameters.lrTopZPosition - stParameters.lrBendingDistance) OR
			mcCartesianZMoveAbsolute.Done THEN
			mcCatcherMoveAbsolute.Execute			:= TRUE;		
			mcCatcherMoveAbsolute.Position			:= stParameters.lrCatcherCatchingPosition;
			mcCatcherMoveAbsolute.Acceleration		:= stParameters.lrCatcherAcceleration;
			mcCatcherMoveAbsolute.Deceleration		:= stParameters.lrCatcherAcceleration;
			mcCatcherMoveAbsolute.Velocity			:= stParameters.lrCatcherSpeed;

//SEL(P190_CapFeeder.stMover2Status.bInPlacePosition, GVL_Recipe.lrCapSorterPreScrewerPickXMover1PositionShow, GVL_Recipe.lrCapSorterPreScrewerPickXMover2PositionShow

			
			//Jedź osią poziomą X na pozycję pick
			mcCartesianYMoveAbsolute.Execute		:= TRUE;
			{warning 'Przerobić, dodać parametry obu pozycji wózków do struktury parametrów, FB_CapPreScrewer.Running --> 624'}
			mcCartesianYMoveAbsolute.Position		:= SEL(bMover1InPickPos, GVL_Recipe.lrCapSorterPreScrewerPickXMover1PositionShow, GVL_Recipe.lrCapSorterPreScrewerPickXMover2PositionShow);
			mcCartesianYMoveAbsolute.Acceleration	:= stParameters.lrPickerAcceleration;
			mcCartesianYMoveAbsolute.Deceleration	:= stParameters.lrPickerAcceleration;
			mcCartesianYMoveAbsolute.Velocity		:= stParameters.lrPickerSpeed;
			//Ustaw obracarkę do pozycji początkowej
			
			mcPreScrewerMoveRelative.Distance		:= -1 * DINT_TO_LREAL(LREAL_TO_DINT(PreScrewerAxisRef.NcToPlc.SetPos) MOD 360); 
			mcPreScrewerMoveRelative.Execute		:= mcPreScrewerMoveRelative.Distance<>0 AND NOT mcPreScrewerMoveRelative.Error;
			mcPreScrewerMoveRelative.Acceleration	:= stParameters.lrScrewAcceleration;
			mcPreScrewerMoveRelative.Deceleration	:= stParameters.lrScrewAcceleration;
			mcPreScrewerMoveRelative.Velocity		:= stParameters.lrScrewSpeed;
			
		END_IF
		IF CartesianZAxisRef.NcToPlc.ActPos > stParameters.lrPlaceZPosition + 20 THEN
			bPlaceDone								:= TRUE;
		END_IF
		IF (*bPlaceDone AND*) mcCartesianYMoveAbsolute.Done AND mcCartesianZMoveAbsolute2.Done AND
			 mcCatcherMoveAbsolute.Done THEN
			 IF mcPreScrewerMoveRelative.Distance=0 OR mcPreScrewerMoveRelative.Done THEN
				mcCartesianYMoveAbsolute.Execute		:= FALSE;
 				mcCartesianZMoveAbsolute.Execute		:= FALSE;
				mcCartesianZMoveAbsolute2.Execute		:= FALSE;
				mcCatcherMoveAbsolute.Execute			:= FALSE;
				mcPreScrewerMoveRelative.Execute		:= FALSE;
				eRunningState				:= E_CapPreScrewer.eDone;
			END_IF
		END_IF
		
		//Dodatkowy przedmuch ssawek
		(*IF (CartesianZAxisRef.NcToPlc.ActPos > (stParameters.lrPlaceZPosition + stParameters.lrHeightAdditionalBlow)) THEN
			bAdditionalBlow							S= NOT tonBlowOFF.IN;	
		
			IF NOT bAdditionalBlow THEN
				bCapsBlowON							R= tonBlowOFF.Q;
			END_IF

			bCapsBlowON								S= bAdditionalBlow;
			bCapBlow1 := bCapBlow2 := bCapBlow3 := bCapBlow4 := bAdditionalBlow;
		END_IF*)
			
	E_CapPreScrewer.eDone:
		mcPreScrewerStop.Execute			:= TRUE;
	
		IF mcPreScrewerStop.Done THEN
			mcPreScrewerStop.Execute			:= FALSE;
			bAdditionalBlow						:= FALSE;
			bCycleNotDone						:= FALSE;
			bCapsBlowON							:= FALSE;
			bPlaceDone							:= TRUE;
			bCycleDone							:= TRUE;
			eState								:= E_Station.eDone;
			eRunningState						:= E_CapPreScrewer.eReady;	
		END_IF	

	(*Cykl nie zakończony - przerwany - chyba nie potrzebny*)
	E_CapPreScrewer.eNotDone:
		bCapsBlowON							:= FALSE;
		eState								:= E_Station.eDone;
		eRunningState						:= E_CapPreScrewer.eReady;




END_CASE

tonCapCatcher(PT := T#60MS);
END_ACTION

ACTION RunningWithFlyingSaw:

tonVacuumWatchdog(PT	:= stParameters.tTimeVacuumWatchdog);
bStopAllowed	:= eRunningState = E_CapPreScrewer.eReady OR eRunningState = E_CapPreScrewer.eVerticalDownToCatchPos;

//Otwieranie chwytaków
//bBottleCatcherCatchTemp		R= CartesianZAxisRef.NcToPlc.ActPos < stParameters.lrGripperOpenPosition;
GVL_VIS.bCapSorterPreScrewerBottleCatcherCatch	:= bBottleCatcherCatchTemp AND bCapSorterPreScrewerBottleCatcherEnableShow;
	
tonWaitInPlacePos(PT	:= stParameters.tWaitInPlacePos);
//tonWaitInPlacePos(PT 	:= T#200MS);
eLastRunningState	:= eRunningState;

CASE eRunningState OF

//====================================
	
	(*Oczekiwanie na wykonanie pojedynczego cyklu*)
	E_CapPreScrewer.eReady:

		
		IF NOT bCycleDone AND NOT bCycleNotDone THEN  
                                      	
			IF bRun THEN 
				fbVirtualAxis.fAcceleration				:= stParameters.lrPickerAcceleration;	
				fbVirtualAxis.fDeceleration				:= stParameters.lrPickerAcceleration;	
				fbVirtualAxis.fJerk						:= stParameters.lrPickerJerk;

				iRejectCase					:= 0;
				bRejectDone					:= FALSE;
				bReject						:= FALSE;
				bTubeReject					:= FALSE;
				
				//Przygotuj do cyklu - otwórz chwytaki
				bCapCatcher1				:= FALSE;
				bCapCatcher2				:= FALSE;
				bCapCatcher3				:= FALSE;
				bCapCatcher4				:= FALSE;
	
				//Wyłącz ssawki
				bCapSucker[1]				:= FALSE;
				bCapSucker[2]				:= FALSE;
				bCapSucker[3]				:= FALSE;
				bCapSucker[4]				:= FALSE;
				//Wyłącz odmuchy
				bCapBlower1					:= FALSE;
				bCapBlower2					:= FALSE;
				bCapBlower3					:= FALSE;
				bCapBlower4					:= FALSE;
				bCapsBlowON					:= FALSE;
				//Otwórz chwytaki słomek
				bStrawCatchersOpen			:= TRUE;
				bStrawCatchersClose			:= FALSE;
				//Cofnij chwytaki słomek
				bStrawCatcherActuatorIn		:= TRUE;
				bStrawCatcherActuatorOut	:= FALSE;
				//Podjedź robotem i chwytakiem słomek w górę jak cofnięty chwytak słomek
				IF tonStrawCatcherIn.Q THEN	
										
					mcCartesianZMoveAbsolute.Execute		:= TRUE;		
					mcCartesianZMoveAbsolute.Position		:= stParameters.lrTopZPosition;
					mcCartesianZMoveAbsolute.Acceleration	:= stParameters.lrPickerAcceleration;
					mcCartesianZMoveAbsolute.Deceleration	:= stParameters.lrPickerAcceleration;
					mcCartesianZMoveAbsolute.Velocity		:= stParameters.lrPickerSpeed;
					
					mcCatcherMoveAbsolute.Execute			:= TRUE;		
					mcCatcherMoveAbsolute.Position			:= stParameters.lrCatcherCatchingPosition;
					mcCatcherMoveAbsolute.Acceleration		:= stParameters.lrCatcherAcceleration;
					mcCatcherMoveAbsolute.Deceleration		:= stParameters.lrCatcherAcceleration;
					mcCatcherMoveAbsolute.Velocity			:= stParameters.lrCatcherSpeed;
					
					//Następny krok
					eRunningState						:= E_CapPreScrewer.ePreparingToPick;
					bCycleNotDone						:= TRUE;
					
				END_IF
				//Reset komendy ruchu osi X
				mcCartesianYMoveAbsolute.Execute		:= FALSE;
				
			END_IF
		END_IF
			
	(*Czekam na pozycję Z w górze i ruszam osią poziomą X na pozycję pobierania i czekam na obie pozycje*)
	E_CapPreScrewer.ePreparingToPick:
		IF (CartesianZAxisRef.NcToPlc.ActPos > stParameters.lrTopZPosition - stParameters.lrBendingDistance) OR
			mcCartesianZMoveAbsolute.Done THEN
			//Jedź osią poziomą X na pozycję pick
			mcCartesianYMoveAbsolute.Execute		:= TRUE;
			mcCartesianYMoveAbsolute.Position		:= stParameters.lrPickYPosition;
			mcCartesianYMoveAbsolute.Acceleration	:= stParameters.lrPickerAcceleration;
			mcCartesianYMoveAbsolute.Deceleration	:= stParameters.lrPickerAcceleration;
			mcCartesianYMoveAbsolute.Velocity		:= stParameters.lrPickerSpeed;
			//Nakrętka pobrana z wózka nr.1
			bMover1InPickPos						:= SEL((stParameters.lrPickYPosition-GVL_Recipe.lrCapSorterPreScrewerPickXMover1PositionShow) <= 0.5, FALSE, TRUE);
			
			//Ustaw obracarkę w pozycji
			mcPreScrewerMoveRelative.Distance		:=  -1 * DINT_TO_LREAL((LREAL_TO_DINT(PreScrewerAxisRef.NcToPlc.SetPos)+diPreSCrewerHomePos) MOD 360);
			mcPreScrewerMoveRelative.Execute		:= mcPreScrewerMoveRelative.Distance<>0;
			mcPreScrewerMoveRelative.Acceleration	:= stParameters.lrScrewAcceleration;
			mcPreScrewerMoveRelative.Deceleration	:= stParameters.lrScrewAcceleration;
			mcPreScrewerMoveRelative.Velocity		:= stParameters.lrScrewSpeed;
		END_IF
		//Jak obie pozycje osiągnięte to wysuń chwytak słomek i następny krok
		IF mcCartesianYMoveAbsolute.Done AND mcCartesianZMoveAbsolute.Done AND mcCatcherMoveAbsolute.Done THEN
			IF mcPreScrewerMoveRelative.Done OR mcPreScrewerMoveRelative.Distance =0 THEN
				//Reset komendy ruchu osi
				mcCartesianYMoveAbsolute.Execute		:= FALSE;
				mcCartesianZMoveAbsolute.Execute		:= FALSE;
				mcPreScrewerMoveRelative.Execute		:= FALSE;
				mcCatcherMoveAbsolute.Execute			:= FALSE;
				//Wysuń chwytaki słomek jesli to potrzebuje recepta        
				bStrawCatcherActuatorIn					:= NOT stParameters.bStrawCatcherON;
				bStrawCatcherActuatorOut				:= stParameters.bStrawCatcherON;    
				//Następny krok
				eRunningState							:= E_CapPreScrewer.ePicking;
			END_IF
		END_IF
		
	
	(*Zjeżdzam na osią pionową Z na pozycję chwytania i załączam ssawki*)		
	E_CapPreScrewer.ePicking:
		//Podjedź robotem w górę	
		mcCartesianZMoveAbsolute.Execute			:= TRUE;		
		mcCartesianZMoveAbsolute.Position			:= stParameters.lrPickZPosition;
		mcCartesianZMoveAbsolute.Acceleration		:= stParameters.lrPickerAcceleration;
		mcCartesianZMoveAbsolute.Deceleration		:= stParameters.lrPickerAcceleration;
		mcCartesianZMoveAbsolute.Velocity			:= stParameters.lrPickerSpeed;
		//Czekam na wykonanie ruchu
		IF mcCartesianZMoveAbsolute.Done THEN
			//Reset komendy ruchu osi
			mcCartesianZMoveAbsolute.Execute		:= FALSE;
			
			//Zeruje rejestry oraz załączanie ssawek
			 FOR i:=1 TO 4 DO
				 bCapSucker[i]						:= stParameters.bPickerActiv[i]; 
				 aCapPresence[i] 					:= FALSE;
			 END_FOR
	
			//Następny krok
			eRunningState							:= E_CapPreScrewer.eVacumCheckPart1;
		END_IF
	
	(*Sprawdzam czy zassane i jazda w górę*)	
	E_CapPreScrewer.eVacumCheckPart1:
		
		tonVacuumWatchdog.IN						:= TRUE;
		
		IF tonSuckedOk[1].Q = stParameters.bPickerActiv[1] AND tonSuckedOk[2].Q = stParameters.bPickerActiv[2]
			AND tonSuckedOk[3].Q = stParameters.bPickerActiv[3] AND tonSuckedOk[4].Q = stParameters.bPickerActiv[4] THEN
			tonVacuumWatchdog.IN					:= FALSE;
		
				FOR i:=1 TO 4 DO
					IF stParameters.bPickerActiv[i] AND stParameters.bStrawCatcherON AND NOT stMoverStatus.stSlotStatus[i].bTubePresent THEN
						bReject								:= TRUE;
						bTubeReject							:= TRUE;
						lrAxisZ_RejectOffset				:= 0.0;
					END_IF

					IF bMover1InPlacePos THEN
						diMover1VacuumRetry[i]		:= 0;
					ELSE
						diMover2VacuumRetry[i]		:= 0;
					END_IF	
				END_FOR 
				
			eRunningState 							:= E_CapPreScrewer.eVacumCheckPart2;
	
		ELSIF tonVacuumWatchdog.Q THEN
		
			FOR i:=1 TO 4 DO
				bCapSucker[i]							:= tonSuckedOk[i].Q;
				
				//robimy odrzut jeżeli zostanie wykryto brak słomki
				IF stParameters.bPickerActiv[i] AND stParameters.bStrawCatcherON AND NOT stMoverStatus.stSlotStatus[i].bTubePresent THEN
					bReject								:= TRUE;
					bTubeReject							:= TRUE;
					lrAxisZ_RejectOffset				:= 0.0;
				END_IF
				
						//Detekcja niepobranej nasadki --> odrzut aktywowany opcjonalnie z receptury
					IF stParameters.bPickerActiv[i] AND NOT tonSuckedOk[i].Q AND NOT stParameters.bVacuumDeactivate THEN
						bReject							:= SEL(stParameters.bRejectON, bReject, TRUE);
						lrAxisZ_RejectOffset			:= SEL(stParameters.bRejectON, lrAxisZ_RejectOffset, 13.0);	//offset dodatkowego zjazdu kartezjanem 
						
						IF bMover1InPlacePos THEN
							diMover1VacuumRetry[i]		:= diMover1VacuumRetry[i] + 1;
						ELSE	
							diMover2VacuumRetry[i]		:= diMover2VacuumRetry[i] + 1;
						END_IF
					ELSIF tonSuckedOk[i].Q OR stParameters.bVacuumDeactivate THEN
						IF 	bMover1InPlacePos THEN
							diMover1VacuumRetry[i]		:= 0;
						ELSE
							diMover2VacuumRetry[i]		:= 0;
						END_IF	
					END_IF	
	    	
			END_FOR
				tonVacuumWatchdog.IN					:= FALSE;
				eRunningState 							:= E_CapPreScrewer.eVacumCheckPart2;
	
		END_IF
		
		
	E_CapPreScrewer.eVacumCheckPart2:	
			
		//Jezeli nie jest przyssana zadna nasadka to pdjezdzamy na poz. ready oraz wystawiamy flage bMissingCaps
		IF bReject THEN
			Reject();
				IF bRejectDone THEN				
					eRunningState						:= E_CapPreScrewer.eReady;	
				END_IF		
		ELSIF NOT tonSuckedOk[1].Q AND NOT tonSuckedOk[2].Q AND NOT tonSuckedOk[3].Q AND NOT tonSuckedOk[4].Q THEN
			bCapSucker[1]							:= FALSE;
			bCapSucker[2]							:= False;
			bCapSucker[3]							:= False;
		    bCapSucker[4]							:= False;	
			mcCartesianZMoveAbsolute.Execute		:= TRUE;		
			mcCartesianZMoveAbsolute.Position		:= stParameters.lrTopZPosition;
			mcCartesianZMoveAbsolute.Acceleration	:= stParameters.lrPickerAcceleration;
			mcCartesianZMoveAbsolute.Deceleration	:= stParameters.lrPickerAcceleration;
			mcCartesianZMoveAbsolute.Velocity		:= stParameters.lrPickerSpeed;
			
			IF mcCartesianZMoveAbsolute.Done THEN
				bMissingCaps						:= TRUE;
				bCycleDone;
				mcCartesianZMoveAbsolute.Execute	:= FALSE;
				eRunningState						:= E_CapPreScrewer.eReady;	
			END_IF
			
		ELSE
			mcCartesianZMoveAbsolute.Execute		:= NOT stParameters.bVacuumDeactivate;		
			mcCartesianZMoveAbsolute.Position		:= stParameters.lrTopZPosition;
			mcCartesianZMoveAbsolute.Acceleration	:= SEL(GVL_Recipe.iCapSorterProductType = 0 ,stParameters.lrPickerAcceleration , 150.0);//stParameters.lrPickerAcceleration;
//			mcCartesianZMoveAbsolute.Acceleration	:= stParameters.lrPickerAcceleration;
			mcCartesianZMoveAbsolute.Deceleration	:= stParameters.lrPickerAcceleration;
			mcCartesianZMoveAbsolute.Velocity		:= stParameters.lrPickerSpeed;
			tonCapCatcher.IN						:= FALSE;
			
			IF mcCartesianZMoveAbsolute.Busy OR stParameters.bVacuumDeactivate THEN
				mcCartesianZMoveAbsolute.Execute		:= FALSE;
				eRunningState 							:= E_CapPreScrewer.eTransferingVertical; 
			END_IF
			
        
		END_IF		
			
			//przepisuje do rejestrów nakretki które kartezjan pobrał
			aCapPresence[1] := bCapSucker[1];
			aCapPresence[2] := bCapSucker[2];
			aCapPresence[3] := bCapSucker[3];
			aCapPresence[4] := bCapSucker[4];						

		
		
	(*Jazda w górę, zamknięcie łapek i załączenie jazdy w bok*)	
	E_CapPreScrewer.eTransferingVertical:
		
		IF NOT bCapSucker[1] OR NOT bCapSucker[2] OR NOT bCapSucker[3] OR NOT bCapSucker[4] THEN
            bCapBlow1						:= NOT bCapSucker[1];
            bCapBlow2						:= NOT bCapSucker[2];
            bCapBlow3						:= NOT bCapSucker[3];
            bCapBlow4						:= NOT bCapSucker[4];						
			bCapsBlowON						:= TRUE;
		END_IF
		
		//Kleją się kulki 
		IF NOT stParameters.bVacuumDeactivate THEN					
			IF CartesianZAxisRef.NcToPlc.ActPos > stParameters.lrPickZPosition + 10.0 THEN
				mcCartesianZMoveAbsolute2.Execute		:= NOT stParameters.bVacuumDeactivate;		
				mcCartesianZMoveAbsolute2.Position		:= stParameters.lrTopZPosition;
				mcCartesianZMoveAbsolute2.Acceleration	:= stParameters.lrPickerAcceleration;
				mcCartesianZMoveAbsolute2.Deceleration	:= stParameters.lrPickerAcceleration;
				mcCartesianZMoveAbsolute2.Velocity		:= stParameters.lrPickerSpeed;
			END_IF
		END_IF


		IF CartesianZAxisRef.NcToPlc.ActPos > stParameters.lrCapCatcherZPosition OR (CartesianZAxisRef.NcToPlc.ActPos > stParameters.lrTopZPosition - stParameters.lrBendingDistance) THEN
			bCapCatcher1							:= TRUE;
			bCapCatcher2							:= true;
			bCapCatcher3							:= true;
			bCapCatcher4							:= true;
			tonCapCatcher.IN						:= stParameters.bVacuumDeactivate;
		END_IF	
		
		mcCartesianZMoveAbsolute.Execute		:= tonCapCatcher.Q;	
		
		//Dodać sprawdzenie czy gotowy chwytak słomek !!!!!
		//Sprawdzenie pozycji osi pionowej Z i czy wysunięty siłownik chwytaka słomek
		IF ((CartesianZAxisRef.NcToPlc.ActPos > stParameters.lrTopZPosition - stParameters.lrBendingDistance) OR
			mcCartesianZMoveAbsolute.Done) AND (tonStrawCatcherOut.Q OR NOT stParameters.bStrawCatcherON) THEN
			//Jedź osią poziomą X na pozycję pick
				mcCartesianZMoveAbsolute2.Execute		:= FALSE;
				bCapsBlowON								:= FALSE;
				eRunningState 							:= E_CapPreScrewer.eTransferingHorizontal;
				tonCapCatcher.IN						:= FALSE;
		END_IF
	
	(*Przejazd w poziomie*)	
	E_CapPreScrewer.eTransferingHorizontal:	
	
			bCapCatcher1							:= TRUE;//bCapSucker1;
			bCapCatcher2							:= TRUE;//bCapSucker2;
			bCapCatcher3							:= TRUE;//bCapSucker3;
			bCapCatcher4							:= TRUE;//bCapSucker4;
	
		mcCartesianYMoveAbsolute.Position			:= stParameters.lrPlaceYPosition;
		mcCartesianYMoveAbsolute.Acceleration		:= stParameters.lrPickerAcceleration;
		mcCartesianYMoveAbsolute.Deceleration		:= stParameters.lrPickerAcceleration;
		mcCartesianYMoveAbsolute.Velocity			:= stParameters.lrPickerSpeed;
		mcCartesianYMoveAbsolute.Execute			:= TRUE;
		
		IF (CartesianYAxisRef.NcToPlc.ActPos > 200.0 (*stParameters.lrPlaceYPosition - stParameters.lrBendingDistance*)) OR
			mcCartesianYMoveAbsolute.Done AND NOT mcCartesianZMoveAbsolute.Execute THEN			

			//Podjedź robotem w dól	
			mcCartesianZMoveAbsolute.Execute			:= TRUE;		
			mcCartesianZMoveAbsolute.Position			:= stParameters.lrCartesianCatchZPosition;
			mcCartesianZMoveAbsolute.Acceleration		:= stParameters.lrPickerAcceleration;
			mcCartesianZMoveAbsolute.Deceleration		:= stParameters.lrPickerAcceleration;
			mcCartesianZMoveAbsolute.Velocity			:= stParameters.lrPickerSpeed;
		END_IF
		
		//Jak obie pozycje osiągnięte 
		IF mcCartesianZMoveAbsolute.Done THEN
			mcCartesianZMoveAbsolute.Execute		:= FALSE;
		END_IF
			
		//Jak ak obie pozycje osiągnięte to zamykamy chwytaki i następny krok
		IF stParameters.bStrawCatcherON AND CartesianYAxisRef.NcToPlc.ActPos >= stParameters.lrPlaceYPosition THEN
			//Zamknij chwytaki słomek
			bStrawCatchersOpen						:= FALSE;
			bStrawCatchersClose						:= TRUE;	
		END_IF
		
			
		IF  mcCartesianYMoveAbsolute.Done AND mcCartesianZMoveAbsolute.Done THEN
			//Reset komendy ruchu osi
			mcCartesianYMoveAbsolute.Execute		:= FALSE;
			mcCartesianZMoveAbsolute.Execute		:= FALSE;
			
				//Ustaw pozycję wirtualnej osi tak samo jak na osi Z
			fbVirtualAxis.fPosition						:=  CartesianZAxisRef.NcToPlc.ActPos;//CartesianZAxisRef.NcToPlc.ActPos - GVL_Recipe.lrCapSorterCapNeckHightShow - GVL_Recipe.lrCapSorterPreScrewerCheckValveShow;
			fbVirtualAxis.SetPosAbsClearLag(bExecute	:= TRUE);
				
				IF fbVirtualAxis.pSetPos.Busy THEN
					//Następny krok
					eRunningState						:= E_CapPreScrewer.eVerticalDownToCatchPos;	
				END_IF
		END_IF		
		
	(*Przejazd w dól do pozycji chwytanija rurki*)		
	E_CapPreScrewer.eVerticalDownToCatchPos:
		fbVirtualAxis.SetPosAbsClearLag(bExecute				:= FALSE);
		
		//Jak ak obie pozycje osiągnięte to zamykamy chwytaki i następny krok
		IF stParameters.bStrawCatcherON THEN
			//Zamknij chwytaki słomek
			bStrawCatchersOpen						:= FALSE;
			bStrawCatchersClose						:= TRUE;	
		END_IF
				
		IF tonPlacePermission.Q AND ((bCapCatcher1 OR NOT bCapCatcher1) AND (bCapCatcher2  OR NOT bCapCatcher2) AND
									(bCapCatcher3  OR NOT bCapCatcher3) AND(bCapCatcher4  OR NOT bCapCatcher4)) AND (tonStrawCatcher1Close.Q OR NOT stParameters.bStrawCatcherON) THEN				
				bCapCatcher1						:= TRUE;
				bCapCatcher2						:= TRUE;
				bCapCatcher3						:= TRUE;
				bCapCatcher4						:= TRUE;						
				eRunningState						:= E_CapPreScrewer.eAxisGearIn;
		END_IF
		
	
	E_CapPreScrewer.eAxisGearIn:
		fbGearInCatcherAxis.Enable						:= stParameters.bStrawCatcherON;
		fbGearInCatcherAxis.GearRatio					:= 1;
		
		fbGearInPos.Execute								:= NOT fbGearInPos.Active;
		fbGearInPos.MasterSyncPosition					:= stParameters.lrCartesianCatchZPosition - (stParameters.lrCapHight - GVL_Recipe.lrCapSorterCapNeckHightShow - GVL_Recipe.lrCapSorterPreScrewerCheckValveShow);//10
		fbGearInPos.SlaveSyncPosition					:= stParameters.lrCartesianCatchZPosition - 15;//15
		
		
		
			IF (fbGearInCatcherAxis.InGear OR NOT stParameters.bStrawCatcherON) AND fbGearInPos.Active AND (tonStrawCatcher1Close.Q (*AND tonStrawCatcher2Close.Q*)
				OR (bStrawCatcherOpen1 AND bStrawCatcherOpen2 AND bStrawCatcherOpen3 AND bStrawCatcherOpen4))  THEN
					fbGearInCatcherAxis.Enable			:= FALSE;
					fbGearInPos.Execute					:= FALSE;
						IF stParameters.bStrawCatcherON THEN
							eRunningState				:= E_CapPreScrewer.ePositionOverBottle;	
							//fbVirtualAxis.fPosition		:= stParameters.lrCartesianCatchZPosition -(CatcherAxisRef.NcToPlc.ActPos - (stParameters.lrBottleHight - stParameters.lrCatcherHightSV - 35));//40mm- offset między łapkami słomek a chwytakami butelek
							lrPreScrewerAxisSavedPosition	:= stParameters.lrCartesianCatchZPosition -(CatcherAxisRef.NcToPlc.ActPos - (stParameters.lrBottleHight - stParameters.lrCatcherHightSV - 35));
							fbVirtualAxis.fPosition		:= (stParameters.LrCheckStrawCatcherActuatorZPosition - (fbGearInPos.SlaveSyncPosition - fbGearInPos.MasterSyncPosition));
						ELSE                            
							eRunningState				:= E_CapPreScrewer.ePlacing;	
						END_IF					
			END_IF		
	
	E_CapPreScrewer.ePositionOverBottle:
		fbVirtualAxis.fVelocity							:= SEL(stParameters.lrCatcherSpeed > 1094.0, stParameters.lrCatcherSpeed, 1094.0 );       						
			
		
		//IF fbVirtualAxis.Axis.NcToPlc.ActPos <= fbVirtualAxis.fPosition	+ 10.0 OR (CatcherAxisRef.NcToPlc.ActPos <= 5.0) THEN
		IF fbVirtualAxis.Axis.NcToPlc.ActPos <= lrPreScrewerAxisSavedPosition	+ 10.0 OR (CatcherAxisRef.NcToPlc.ActPos <= 5.0) THEN
			fbGearInCatcherAxis.GearRatio				:= 0.0000000000000000000000000000000000000000000000000000000000001;		
			fbGearOutCatcherAxis.Execute				:= CatcherAxisRef.Status.Coupled;
			mcCatcherStop.Execute						:= 	NOT CatcherAxisRef.Status.Coupled ;
			bVirtualMove								:= FALSE;
		ELSE
			bVirtualMove								:= TRUE;	
		END_IF 
		
		IF NOT CatcherAxisRef.Status.Coupled AND (NOT CatcherAxisRef.Status.Moving OR mcCatcherStop.Busy) THEN
			eRunningState							:= E_CapPreScrewer.eCatching;	
		END_IF
	
	
	//Sprawdzanie czy chwytaki zamknięte i opuszczenie chwytaków do dolnej pozycji
	E_CapPreScrewer.eCatching:
		fbVirtualAxis.fPosition							:= (stParameters.LrCheckStrawCatcherActuatorZPosition - (fbGearInPos.SlaveSyncPosition - fbGearInPos.MasterSyncPosition));// - stParameters.lrStrawInsertDistance);	//Pozycja sprawdzania cofnięcia krabów
		fbVirtualAxis.fVelocity							:= SEL(stParameters.lrCatcherSpeed > 1094.0, stParameters.lrCatcherSpeed, 1094.0 );       						
		bVirtualMove									:= TRUE;					
	
			//Otwórz chwytaki słomek
		IF CartesianZAxisRef.NcToPlc.ActPos <= stParameters.lrStrawCatcherZPosition THEN		
			bStrawCatchersOpen							:= TRUE;
			bStrawCatchersClose							:= FALSE;
			
				IF tonStrawCatcher1Open.Q AND tonStrawCatcher2Open.Q AND tonStrawCatcher3Open.Q AND tonStrawCatcher4Open.Q THEN																				
					//Cofnij chwytaki słomek
					bStrawCatcherActuatorIn				:= TRUE;
					bStrawCatcherActuatorOut			:= FALSE;				
				END_IF	
		ELSE
			fbGearInCatcherAxis.GearRatio				:= F_Scaling((CatcherAxisRef.NcToPlc.ActPos*10), 0.0, 10.0, 0.0, 1.0);
			fbGearInCatcherAxis.GearRatio				:= SEL(fbGearInCatcherAxis.GearRatio>1.0, fbGearInCatcherAxis.GearRatio, 1.0);	
		END_IF		
						
				IF bStrawCatcherIn THEN
					fbGearOutCatcherAxis.Execute		:= FALSE;
					mcCatcherStop.Execute				:= FALSE;
					bVirtualMove						:= FALSE;	
					eRunningState						:= E_CapPreScrewer.ePlacing;
				END_IF		
			
		//END_IF
	


	
	//Czekaj aż chwytak słomek dojedzie do dołu i zacznij ruch osi pionowej Z
	E_CapPreScrewer.ePlacing:		
		IF stParameters.lrScrewFinding > 0 THEN
			eRunningState								:= E_CapPreScrewer.eFinding;
		ELSE
			lrPreScrewerAxisSavedPosition				:= PreScrewerAxisRef.NcToPlc.ActPos;	//zapisywanie pozycji przed zakrecaniem		
			fbVirtualAxis.fPosition						:= SEL(stParameters.bStrawCatcherON, stParameters.lrScrewerStartZPosition, stParameters.lrScrewerStartZPosition - (fbGearInPos.SlaveSyncPosition - fbGearInPos.MasterSyncPosition));//stParameters.lrPlaceZPosition, stParameters.lrPlaceZPosition - (fbGearInPos.SlaveSyncPosition - fbGearInPos.MasterSyncPosition));//stParameters.lrStrawInsertDistance);
			fbVirtualAxis.fVelocity						:= SEL(stParameters.lrCatcherSpeed > 1094.0, stParameters.lrCatcherSpeed, 1094.0 );    
			bVirtualMove								:= TRUE;
			
			eRunningState								:= E_CapPreScrewer.ePreScrewing;
		END_IF
	
	E_CapPreScrewer.eFinding:
		fbVirtualAxis.fPosition							:= SEL(stParameters.bStrawCatcherON, stParameters.lrScrewerStartZPosition, stParameters.lrScrewerStartZPosition - (fbGearInPos.SlaveSyncPosition - fbGearInPos.MasterSyncPosition));// stParameters.lrScrewerStartZPosition-stParameters.lrStrawInsertDistance);
		fbVirtualAxis.fVelocity							:= SEL(stParameters.lrCatcherSpeed > 1094.0, stParameters.lrCatcherSpeed, 1094.0 );
		fbVirtualAxis.fAcceleration						:= stParameters.lrCatcherAcceleration; 
		fbVirtualAxis.fDeceleration						:= stParameters.lrCatcherAcceleration; 
		fbVirtualAxis.fJerk								:= stParameters.lrCatcherJerk;        		
			                                            
		bVirtualMove									:= TRUE;
		                                                
			IF ABS(fbVirtualAxis.Axis.NcToPlc.ActPos - fbVirtualAxis.fPosition) <= 0.5 THEN              
				bCapSucker[1]								:= FALSE;
				bCapSucker[2]								:= FALSE;
				bCapSucker[3]								:= FALSE;
				bCapSucker[4]								:= FALSE;
    	                                                
				mcPreScrewerMoveRelative.Distance		:= stParameters.lrScrewFinding * -1.0;
				mcPreScrewerMoveRelative.Acceleration	:= stParameters.lrScrewAcceleration;
				mcPreScrewerMoveRelative.Deceleration	:= stParameters.lrScrewAcceleration;
				mcPreScrewerMoveRelative.Velocity		:= stParameters.lrScrewSpeed;
				mcPreScrewerMoveRelative.Execute		:= TRUE;
			END_IF
			
					IF mcPreScrewerMoveRelative.Done OR ABS(PreScrewerAxisRef.NcToPlc.PosDiff) > 60.0 OR mcPreScrewerMoveRelative.Error THEN
						bVirtualMove							:= FALSE;
						mcPreScrewerMoveRelative.Execute		:= FALSE;
						eRunningState							:= E_CapPreScrewer.ePreScrewing;
					END_IF	
	
	E_CapPreScrewer.ePreScrewing:

	IF ABS(fbVirtualAxis.Axis.NcToPlc.ActPos - fbVirtualAxis.fPosition)<=0.1 THEN
		bVirtualMove											:= FALSE;
		
		IF NOT	CartesianZAxisRef.Status.Coupled THEN
			eRunningState				:= E_CapPreScrewer.eScrewing;
			mcCartesianZStop.Execute	:= FALSE;
			fbGearOutAxisZ.Execute		:= FALSE;
		ELSE
			fbGearOutAxisZ.Execute		:= TRUE;
			mcCartesianZStop.Execute	:= CartesianZAxisRef.Status.Moving;
		END_IF	
	END_IF
		
	
	
	E_CapPreScrewer.eScrewing:
	
			fbGearInAxisZ_Screwer.Execute			:= NOT CartesianZAxisRef.Status.Coupled AND NOT mcCartesianZStop.Busy;
			fbGearInAxisZ_Screwer.RatioNumerator 	:= (GVL_Recipe.lrCapSorterPreScrewerThreadPitchShow	* GVL_Recipe.lrCapSorterPreScrewerMultipleStartThreadShow * (-1));
			fbGearInAxisZ_Screwer.RatioDenominator	:= 360;
		
			IF CartesianZAxisRef.Status.Coupled THEN	//+8
						mcPreScrewerMoveRelative.Execute		:= TRUE;
						mcPreScrewerMoveRelative.Distance		:= stParameters.lrScrewDistance;
						mcPreScrewerMoveRelative.Acceleration	:= stParameters.lrScrewAcceleration;
						mcPreScrewerMoveRelative.Deceleration	:= stParameters.lrScrewAcceleration;
						mcPreScrewerMoveRelative.Velocity		:= stParameters.lrScrewSpeed;	
						eRunningState							:= E_CapPreScrewer.eFinished;	
			END_IF
	
	//Kończenie cyklu zakręcania - otwarcie chwytaka
	E_CapPreScrewer.eFinished:		
	
		IF PreScrewerAxisRef.NcToPlc.PosDiff > 100.0 OR mcPreScrewerMoveRelative.Done THEN
//			bBottleCatcherCatchTemp							:= FALSE;	
			bCapCatcher1									:= FALSE;
		 	bCapCatcher2									:= FALSE;
		 	bCapCatcher3									:= FALSE;
		 	bCapCatcher4									:= FALSE;
			mcPreScrewerMoveRelative.Execute				:= FALSE;
			bVirtualMove									:= FALSE;
			bCapBlow1										:= bCapSucker[1];
            bCapBlow2										:= bCapSucker[2];
            bCapBlow3										:= bCapSucker[3];
            bCapBlow4										:= bCapSucker[4];
			bCapSucker[1]									:= FALSE;
			bCapSucker[2]									:= FALSE;
			bCapSucker[3]									:= FALSE;
			bCapSucker[4]									:= FALSE;								
			
				IF PreScrewerAxisRef.Status.Moving THEN
					mcPreScrewerStop.Execute				:=	 TRUE;					
				ELSE
					lrAxisZSavedPosition					:= CartesianZAxisRef.NcToPlc.ActPos;
					mcPreScrewerStop.Execute				:= FALSE;
					fbGearInCatcherAxis.Enable				:= FALSE;
					eRunningState							:= E_CapPreScrewer.eGearOut;
				END_IF	
		END_IF
		
	E_CapPreScrewer.eGearOut:
		fbGearOutAxisZ.Execute								:= TRUE;
		fbGearOutCatcherAxis.Execute						:= TRUE;
	
			IF NOT CartesianZAxisRef.Status.Coupled AND NOT CatcherAxisRef.Status.Coupled THEN
				fbGearOutAxisZ.Execute						:= FALSE;
				fbGearOutCatcherAxis.Execute				:= FALSE;
				eRunningState								:= E_CapPreScrewer.eReturning1;
			END_IF
	
	//Powrót na górną pozycję
	E_CapPreScrewer.eReturning1:
	
		tonWaitInPlacePos.IN						:= TRUE;
		mcPreScrewerStop.Execute					:= TRUE;		

		IF tonWaitInPlacePos.Q THEN
			

		
			tonWaitInPlacePos.IN					:= FALSE;
//			bBottleCatcherCatchTemp					:= FALSE;		
			mcPreScrewerStop.Execute				:= FALSE;
			mcCartesianZMoveAbsolute.Execute		:= TRUE;
			mcCartesianZMoveAbsolute.Position		:= stParameters.lrTopZPosition;
			mcCartesianZMoveAbsolute.Acceleration	:= SEL(GVL_Recipe.iCapSorterProductType = 0 ,stParameters.lrPickerAcceleration , 150.0);
//			mcCartesianZMoveAbsolute.Acceleration	:= stParameters.lrPickerAcceleration;
			mcCartesianZMoveAbsolute.Deceleration	:= stParameters.lrPickerAcceleration;
			mcCartesianZMoveAbsolute.Velocity		:= stParameters.lrPickerSpeed;
			
			IF mcCartesianZMoveAbsolute.Busy THEN
				mcCartesianZMoveAbsolute.Execute		:= FALSE;
				eRunningState							:= E_CapPreScrewer.eReturning2;
			END_IF
			
		END_IF
		

		
	//Powrót po osi X	
	E_CapPreScrewer.eReturning2:
		bBottleCatcherCatchTemp					:= FALSE;
		bCapsBlowON								:= CartesianZAxisRef.NcToPlc.ActPos > lrAxisZSavedPosition + 10.0;
		
		IF CartesianZAxisRef.NcToPlc.ActPos > stParameters.lrScrewerStartZPosition + 15.0 THEN
			mcCartesianZMoveAbsolute2.Execute		:= TRUE;
			mcCartesianZMoveAbsolute2.Position		:= stParameters.lrTopZPosition;
			mcCartesianZMoveAbsolute2.Acceleration	:= stParameters.lrPickerAcceleration;
			mcCartesianZMoveAbsolute2.Deceleration	:= stParameters.lrPickerAcceleration;
			mcCartesianZMoveAbsolute2.Velocity		:= stParameters.lrPickerSpeed;			
		END_IF
	
		IF (CartesianZAxisRef.NcToPlc.ActPos > stParameters.lrTopZPosition - stParameters.lrBendingDistance) OR
			mcCartesianZMoveAbsolute.Done THEN
			mcCatcherMoveAbsolute.Execute			:= TRUE;		
			mcCatcherMoveAbsolute.Position			:= stParameters.lrCatcherCatchingPosition;
			mcCatcherMoveAbsolute.Acceleration		:= stParameters.lrCatcherAcceleration;
			mcCatcherMoveAbsolute.Deceleration		:= stParameters.lrCatcherAcceleration;
			mcCatcherMoveAbsolute.Velocity			:= stParameters.lrCatcherSpeed;

//SEL(P190_CapFeeder.stMover2Status.bInPlacePosition, GVL_Recipe.lrCapSorterPreScrewerPickXMover1PositionShow, GVL_Recipe.lrCapSorterPreScrewerPickXMover2PositionShow

			
			//Jedź osią poziomą X na pozycję pick
			mcCartesianYMoveAbsolute.Execute		:= TRUE;
			{warning 'Przerobić, dodać parametry obu pozycji wózków do struktury parametrów, FB_CapPreScrewer.Running --> 624'}
			mcCartesianYMoveAbsolute.Position		:= SEL(bMover1InPickPos, GVL_Recipe.lrCapSorterPreScrewerPickXMover1PositionShow, GVL_Recipe.lrCapSorterPreScrewerPickXMover2PositionShow);
			mcCartesianYMoveAbsolute.Acceleration	:= stParameters.lrPickerAcceleration;
			mcCartesianYMoveAbsolute.Deceleration	:= stParameters.lrPickerAcceleration;
			mcCartesianYMoveAbsolute.Velocity		:= stParameters.lrPickerSpeed;
			//Ustaw obracarkę do pozycji początkowej
			
			mcPreScrewerMoveRelative.Distance		:= -1 * DINT_TO_LREAL(LREAL_TO_DINT(PreScrewerAxisRef.NcToPlc.SetPos) MOD 360); 
			mcPreScrewerMoveRelative.Execute		:= mcPreScrewerMoveRelative.Distance<>0 AND NOT mcPreScrewerMoveRelative.Error;
			mcPreScrewerMoveRelative.Acceleration	:= stParameters.lrScrewAcceleration;
			mcPreScrewerMoveRelative.Deceleration	:= stParameters.lrScrewAcceleration;
			mcPreScrewerMoveRelative.Velocity		:= stParameters.lrScrewSpeed;
			
		END_IF
		IF CartesianZAxisRef.NcToPlc.ActPos > stParameters.lrPlaceZPosition + 20 THEN
			bPlaceDone								:= TRUE;
		END_IF
		IF (*bPlaceDone AND*) mcCartesianYMoveAbsolute.Done AND mcCartesianZMoveAbsolute2.Done AND
			 mcCatcherMoveAbsolute.Done THEN
			 IF mcPreScrewerMoveRelative.Distance=0 OR mcPreScrewerMoveRelative.Done THEN
				mcCartesianYMoveAbsolute.Execute		:= FALSE;
 				mcCartesianZMoveAbsolute.Execute		:= FALSE;
				mcCartesianZMoveAbsolute2.Execute		:= FALSE;
				mcCatcherMoveAbsolute.Execute			:= FALSE;
				mcPreScrewerMoveRelative.Execute		:= FALSE;
				eRunningState				:= E_CapPreScrewer.eDone;
			END_IF
		END_IF
		
		//Dodatkowy przedmuch ssawek
		(*IF (CartesianZAxisRef.NcToPlc.ActPos > (stParameters.lrPlaceZPosition + stParameters.lrHeightAdditionalBlow)) THEN
			bAdditionalBlow							S= NOT tonBlowOFF.IN;	
		
			IF NOT bAdditionalBlow THEN
				bCapsBlowON							R= tonBlowOFF.Q;
			END_IF

			bCapsBlowON								S= bAdditionalBlow;
			bCapBlow1 := bCapBlow2 := bCapBlow3 := bCapBlow4 := bAdditionalBlow;
		END_IF*)
			
	E_CapPreScrewer.eDone:
		mcPreScrewerStop.Execute			:= TRUE;
	
		IF mcPreScrewerStop.Done THEN
			mcPreScrewerStop.Execute			:= FALSE;
			bAdditionalBlow						:= FALSE;
			bCycleNotDone						:= FALSE;
			bCapsBlowON							:= FALSE;
			bPlaceDone							:= TRUE;
			bCycleDone							:= TRUE;
			eState								:= E_Station.eDone;
			eRunningState						:= E_CapPreScrewer.eReady;	
		END_IF	

	(*Cykl nie zakończony - przerwany - chyba nie potrzebny*)
	E_CapPreScrewer.eNotDone:
		bCapsBlowON							:= FALSE;
		eState								:= E_Station.eDone;
		eRunningState						:= E_CapPreScrewer.eReady;




END_CASE

tonCapCatcher(PT := T#60MS);
END_ACTION

ACTION Signals:
rtChoseRecipe(CLK := stCommandsIn.bChoseRecipe);
rtAxisZMoving(CLK := CartesianZAxisRef.Status.Moving);
bHomingWithoutJiesang	R= rtChoseRecipe.Q;

//Filtry sygnałów z czujników 
tonSuckedOk[1](IN:=bCapSucker[1] AND (stParameters.bVacuumDeactivate OR bCapSuckerVacumOk1), PT:=T#4MS);
tonSuckedOk[2](IN:=bCapSucker[2] AND (stparameters.bvacuumDeactivate OR bCapSuckerVacumOk2), PT:=T#4MS);
tonSuckedOk[3](IN:=bCapSucker[3] AND (stparameters.bvacuumDeactivate OR bCapSuckerVacumOk3), PT:=T#4MS);
tonSuckedOk[4](IN:=bCapSucker[4] AND (stparameters.bvacuumDeactivate OR bCapSuckerVacumOk4), PT:=T#4MS);

tonStrawCatcherIn(In:=bStrawCatcherIn, PT:=T#4MS); 
tonStrawCatcherOut(In:=bStrawCatcherOut, PT:=T#4MS);

tonStrawCatcher1Open(In:=  bStrawCatcherOpen1, PT:=T#0MS); 
tonStrawCatcher2Open(In:=  bStrawCatcherOpen2, PT:=T#0MS); 
tonStrawCatcher3Open(In:=  bStrawCatcherOpen3, PT:=T#0MS); 
tonStrawCatcher4Open(In:=  bStrawCatcherOpen4, PT:=T#0MS); 

tonStrawCatcher1Close(In:=NOT bStrawCatcherOpen1 OR bStrawCatchersClose, PT:=T#120MS); 
tonStrawCatcher2Close(In:=NOT bStrawCatcherOpen2, PT:=T#0MS); 
tonStrawCatcher3Close(In:=NOT bStrawCatcherOpen3, PT:=T#0MS); 
tonStrawCatcher4Close(In:=NOT bStrawCatcherOpen4, PT:=T#0MS); 	

tonCapCatcher1Open(IN:= NOT bCapCatcher1, PT := T#50MS);

tonBlowOFF.PT := SEL(eRunningState = E_CapPreScrewer.eTransferingVertical, T#250MS, T#2S);
tonBlowOFF(In:=bCapsBlowON); 	//250ms //dp bylo 50
tonBlowerON[1](In:=bCapsBlowON, PT:=T#0MS); //timery na załączanie kolejnych cewek
tonBlowerON[2](In:=bCapsBlowON, PT:=T#4MS); (*T#15MS*)
tonBlowerON[3](In:=bCapsBlowON, PT:=T#8MS); 
tonBlowerON[4](In:=bCapsBlowON, PT:=T#12MS);

bCapBlower1 			:= (*tonBlowerON[1].Q AND*) bCapsBlowON AND NOT tonBlowOFF.Q AND (bCapBlow1 (*OR aCapPresence[1]*));
bCapBlower2 			:= (*tonBlowerON[2].Q AND*) bCapsBlowON AND NOT tonBlowOFF.Q AND (bCapBlow2 (*OR aCapPresence[2]*));
bCapBlower3 			:= (*tonBlowerON[3].Q AND*) bCapsBlowON AND NOT tonBlowOFF.Q AND (bCapBlow3 (*OR aCapPresence[3]*));
bCapBlower4 			:= (*tonBlowerON[4].Q AND*) bCapsBlowON AND NOT tonBlowOFF.Q AND (bCapBlow4 (*OR aCapPresence[4]*));
	
tonPlacePermission(IN 	:= bPlacePermission, PT:=T#30MS); 
rtPlacePermission(CLk 	:= tonPlacePermission.Q);
rtRun(CLK	:= bRun);
//Żądanie zamknięcia chwytaków
IF rtPlacePermission.Q THEN
	bBottleCatcherCatchTemp			:= TRUE;
END_IF

//Przewidywane zatrzymanie, wymuś bazowanie jezeli kartezjan nie bedzie na tych pozycjach!!!!!
bCartesianInReadyPos	:= (eRunningState = E_CapPreScrewer.eReady) OR
							(eRunningState = E_CapPreScrewer.eVerticalDownToCatchPos);
	
//Flagi pomocnicze dla bazowania- AxisY jest na pozycji
bAxisYInPosition	:= ABS(mcCartesianYMoveAbsolute.Position - CartesianYAxisRef.NcToPlc.ActPos) < 10.0;

//Flagi pomocnicze dla bazowania- AxisZ jest na pozycji 1
bAxisZInPosition1 := NOT CartesianZAxisRef.Status.Moving AND ABS(mcCartesianZMoveAbsolute.Position - CartesianZAxisRef.NcToPlc.ActPos) < 10.0;

//Flagi pomocnicze dla bazowania- AxisZ jest na pozycji 2
bAxisZInPosition2	:= NOT CartesianZAxisRef.Status.Moving AND ABS(mcCartesianZMoveAbsolute2.Position - CartesianZAxisRef.NcToPlc.ActPos) < 10.0;

//Oś Z jest na pozycji
bAxisZInPosition := bAxisZInPosition1 OR bAxisZInPosition2;
															
IF tonBlowOFF.Q THEN
	bCapsBlowON 							:= FALSE;
	bCapBlow1								:= FALSE;
	bCapBlow2								:= FALSE;
	bCapBlow3								:= FALSE;
	bCapBlow4								:= FALSE;
END_IF

bAxisYSafePos			:= CartesianYAxisRef.NcToPlc.ActPos > 250.0;
bCartesianSafePos			:= (CartesianZAxisRef.NcToPlc.ActPos >= 310.0) OR bAxisYSafePos;

//Monitoring utraconych nasadek, sprawdzamy tylko gdy odjeżdżamy do poz. place oraz mamy zamknąć wings'y
IF eRunningState > 5 AND eRunningState < 30 THEN
	bCapLost[1]								:= NOT bCapCatcher1  AND stParameters.bPickerActiv[1]; 
	bCapLost[2]								:= NOT bCapCatcher2  AND stParameters.bPickerActiv[2]; 
	bCapLost[3]								:= NOT bCapCatcher3  AND stParameters.bPickerActiv[3]; 
	bCapLost[4]								:= NOT bCapCatcher4  AND stParameters.bPickerActiv[4]; 
	bAnyCapLost								:= bCapLost[1] OR bCapLost[2] OR bCapLost[3] OR bCapLost[4];
ELSE
	bCapLost[1]								:= FALSE;
    bCapLost[2]								:= False;
    bCapLost[3]								:= False;
    bCapLost[4]								:= False;
    bAnyCapLost								:= False;
END_IF

bAnyCapPresence		:= (bCapSuckerVacumOk1 OR bCapCatcher1 OR bCapSuckerVacumOk2 OR bCapCatcher2 OR 
						bCapSuckerVacumOk3 OR bCapCatcher3 OR bCapSuckerVacumOk4 OR bCapCatcher4);

bAxisZInHomePos 	:= ABS(CartesianZAxisRef.NcToPlc.ActPos - 420.0) <= 1.0;
bAxisZInTopPos		:= ABS(CartesianZAxisRef.NcToPlc.ActPos - stParameters.lrTopZPosition) <= 1.0;
bAxisYInHomePos		:= ABS(CartesianYAxisRef.NcToPlc.ActPos - stParameters.lrPickYPosition) <= 1.0;
bStrawCatcherLiftInHomePos := tonStrawCatcherLiftInHomePos.Q;
bCartesianInHomePos	:= bAxisZInHomePos AND bAxisYInHomePos;
bCartesianInTopPos  := bAxisZInTopPos AND bAxisYInHomePos;

//Kąt początkowy zakręcarki
diPreSCrewerHomePos	:= SEL(GVL_Recipe.bCapSorterPreScrewerPoundedInCap, 0, 90);

//Monitorowanie momentu na osiach
CartesianYAxisRef.NcToPlc.ActTorque;
CartesianZAxisRef.NcToPlc.ActTorque;
CatcherAxisRef.NcToPlc.ActTorque;


bCapScrewed		:= (eLastRunningState = E_CapPreScrewer.eFinding OR eLastRunningState = E_CapPreScrewer.eFindingStop
					OR eLastRunningState = E_CapPreScrewer.eScrewing OR eLastRunningState = E_CapPreScrewer.eFinished
					OR eLastRunningState = E_CapPreScrewer.eReturning1);


tonStrawCatcherLiftInHomePos(IN := ABS(GVL_VIS.lrCapSorterPreScrewerCatcherStationHeightCV-stParameters.lrCatcherHightSV) <= 1.0, PT := T#3S);

FOR i:=1 TO 4 DO
	arrVacuumStatus[i] := tonSuckedOk[i].Q OR (NOT bCapSucker[i] AND NOT stParameters.bPickerActiv[i]);
END_FOR


bAllSlotsVacuumStatus	:= arrVacuumStatus[1] AND arrVacuumStatus[2] AND arrVacuumStatus[3] AND arrVacuumStatus[4];
END_ACTION

ACTION Simulation:
tonVacuumWatchdog(PT	:= stParameters.tTimeVacuumWatchdog);
bStopAllowed	:= iSimulationCase = 0;

CASE iSimulationCase OF
	0:
			IF NOT bCycleDone AND NOT bCycleNotDone THEN  
				IF bRun THEN 
				iRejectCase					:= 0;
				bRejectDone					:= FALSE;
				bReject						:= FALSE;
				bTubeReject					:= FALSE;
				
				//Przygotuj do cyklu - otwórz chwytaki
				bCapCatcher1				:= FALSE;
				bCapCatcher2				:= FALSE;
				bCapCatcher3				:= FALSE;
				bCapCatcher4				:= FALSE;
	
				//Wyłącz ssawki
				bCapSucker[1]				:= FALSE;
				bCapSucker[2]				:= FALSE;
				bCapSucker[3]				:= FALSE;
				bCapSucker[4]				:= FALSE;
				//Wyłącz odmuchy
				bCapBlower1					:= FALSE;
				bCapBlower2					:= FALSE;
				bCapBlower3					:= FALSE;
				bCapBlower4					:= FALSE;
				bCapsBlowON					:= FALSE;
				//Otwórz chwytaki słomek
				bStrawCatchersOpen			:= TRUE;
				bStrawCatchersClose			:= FALSE;
				//Cofnij chwytaki słomek
				bStrawCatcherActuatorIn		:= TRUE;
				bStrawCatcherActuatorOut	:= FALSE;
				
					IF tonStrawCatcherIn.Q THEN	
											
						mcCartesianZMoveAbsolute.Execute		:= TRUE;		
						mcCartesianZMoveAbsolute.Position		:= stParameters.lrTopZPosition;
						mcCartesianZMoveAbsolute.Acceleration	:= stParameters.lrPickerAcceleration;
						mcCartesianZMoveAbsolute.Deceleration	:= stParameters.lrPickerAcceleration;
						mcCartesianZMoveAbsolute.Velocity		:= stParameters.lrPickerSpeed;
						
						mcCatcherMoveAbsolute.Execute			:= TRUE;		
						mcCatcherMoveAbsolute.Position			:= stParameters.lrCatcherCatchingPosition;
						mcCatcherMoveAbsolute.Acceleration		:= stParameters.lrCatcherAcceleration;
						mcCatcherMoveAbsolute.Deceleration		:= stParameters.lrCatcherAcceleration;
						mcCatcherMoveAbsolute.Velocity			:= stParameters.lrCatcherSpeed;
						
						//Następny krok
						iSimulationCase		:= 10;
						
					END_IF
				//Reset komendy ruchu osi X
				mcCartesianYMoveAbsolute.Execute		:= FALSE;
				
			END_IF
		END_IF	
				
		10:
			IF (CartesianZAxisRef.NcToPlc.ActPos > stParameters.lrTopZPosition - stParameters.lrBendingDistance) OR
				mcCartesianZMoveAbsolute.Done THEN
				//Jedź osią poziomą X na pozycję pick
				mcCartesianYMoveAbsolute.Execute		:= TRUE;
				mcCartesianYMoveAbsolute.Position		:= stParameters.lrPickYPosition;
				mcCartesianYMoveAbsolute.Acceleration	:= stParameters.lrPickerAcceleration;
				mcCartesianYMoveAbsolute.Deceleration	:= stParameters.lrPickerAcceleration;
				mcCartesianYMoveAbsolute.Velocity		:= stParameters.lrPickerSpeed;
				//Nakrętka pobrana z wózka nr.1
				bMover1InPickPos						:= SEL((stParameters.lrPickYPosition-GVL_Recipe.lrCapSorterPreScrewerPickXMover1PositionShow) <= 0.5, FALSE, TRUE);
				
				//Ustaw obracarkę w pozycji
				mcPreScrewerMoveRelative.Distance		:=  -1 * DINT_TO_LREAL((LREAL_TO_DINT(PreScrewerAxisRef.NcToPlc.SetPos)+diPreSCrewerHomePos) MOD 360);
				mcPreScrewerMoveRelative.Execute		:= mcPreScrewerMoveRelative.Distance<>0;
				mcPreScrewerMoveRelative.Acceleration	:= stParameters.lrScrewAcceleration;
				mcPreScrewerMoveRelative.Deceleration	:= stParameters.lrScrewAcceleration;
				mcPreScrewerMoveRelative.Velocity		:= stParameters.lrScrewSpeed;
			END_IF
			//Jak obie pozycje osiągnięte to wysuń chwytak słomek i następny krok
			IF mcCartesianYMoveAbsolute.Done AND mcCartesianZMoveAbsolute.Done AND mcCatcherMoveAbsolute.Done THEN
				IF mcPreScrewerMoveRelative.Done OR mcPreScrewerMoveRelative.Distance =0 THEN
					//Reset komendy ruchu osi
					mcCartesianYMoveAbsolute.Execute		:= FALSE;
					mcCartesianZMoveAbsolute.Execute		:= FALSE;
					mcPreScrewerMoveRelative.Execute		:= FALSE;
					mcCatcherMoveAbsolute.Execute			:= FALSE;
					//Wysuń chwytaki słomek jesli to potrzebuje recepta        
					bStrawCatcherActuatorIn					:= NOT stParameters.bStrawCatcherON;
					bStrawCatcherActuatorOut				:= stParameters.bStrawCatcherON;    
					//Następny krok
					iSimulationCase		:= 20;
				END_IF
			END_IF		
	
		20:
				mcCartesianZMoveAbsolute.Execute			:= TRUE;		
				mcCartesianZMoveAbsolute.Position			:= stParameters.lrPickZPosition;
				mcCartesianZMoveAbsolute.Acceleration		:= stParameters.lrPickerAcceleration;
				mcCartesianZMoveAbsolute.Deceleration		:= stParameters.lrPickerAcceleration;
				mcCartesianZMoveAbsolute.Velocity			:= stParameters.lrPickerSpeed;
					
			//Czekam na wykonanie ruchu
			IF mcCartesianZMoveAbsolute.Done THEN
				//Reset komendy ruchu osi
				mcCartesianZMoveAbsolute.Execute		:= FALSE;
				
				//Zeruje rejestry oraz załączanie ssawek
				 FOR i:=1 TO 4 DO
					 bCapSucker[i]						:= TRUE; 
					 aCapPresence[i] 					:= FALSE;					 
						IF stParameters.bPickerActiv[i] AND stParameters.bStrawCatcherON AND NOT stMoverStatus.stSlotStatus[i].bTubePresent THEN
							bReject								:= TRUE;
							bTubeReject							:= TRUE;
							lrAxisZ_RejectOffset				:= 0.0;
						END_IF
				 END_FOR
	    	
				//Następny krok
				iSimulationCase		:= 30;
			END_IF
	
		30:
			tonVacuumWatchdog.IN						:= TRUE;
		
			IF (tonSuckedOk[1].Q = stParameters.bPickerActiv[1] AND tonSuckedOk[2].Q = stParameters.bPickerActiv[2]
				AND tonSuckedOk[3].Q = stParameters.bPickerActiv[3] AND tonSuckedOk[4].Q = stParameters.bPickerActiv[4]) OR tonVacuumWatchdog.Q THEN
				tonVacuumWatchdog.IN					:= FALSE;
			
					FOR i:=1 TO 4 DO
						IF bMover1InPlacePos THEN
							diMover1VacuumRetry[i]		:= 0;
						ELSE
							diMover2VacuumRetry[i]		:= 0;
						END_IF	
					END_FOR 
					
				iSimulationCase		:= 40;
			END_IF	
			
		35:
			IF bReject THEN
				Reject();
				IF bRejectDone THEN				
					iSimulationCase					:= 0;	
				END_IF		
			ELSE
				iSimulationCase						:= 40;	
			END_IF	

		40:
			mcCartesianZMoveAbsolute.Execute		:= NOT stParameters.bVacuumDeactivate;		
			mcCartesianZMoveAbsolute.Position		:= stParameters.lrTopZPosition;
			mcCartesianZMoveAbsolute.Acceleration	:= SEL(GVL_Recipe.iCapSorterProductType = 0 ,stParameters.lrPickerAcceleration , 70.0);//stParameters.lrPickerAcceleration;
			mcCartesianZMoveAbsolute.Deceleration	:= stParameters.lrPickerAcceleration;
			mcCartesianZMoveAbsolute.Velocity		:= stParameters.lrPickerSpeed;
			tonCapCatcher.IN						:= FALSE;
			
				//przepisuje do rejestrów nakretki które kartezjan pobrał
			aCapPresence[1] := bCapSucker[1];
			aCapPresence[2] := bCapSucker[2];
			aCapPresence[3] := bCapSucker[3];
			aCapPresence[4] := bCapSucker[4];	
			
			IF mcCartesianZMoveAbsolute.Busy OR stParameters.bVacuumDeactivate THEN
				mcCartesianZMoveAbsolute.Execute		:= FALSE;
				iSimulationCase		:= 50;
			END_IF
		
		50:
				//Kleją się kulki 
			IF NOT stParameters.bVacuumDeactivate THEN					
				IF CartesianZAxisRef.NcToPlc.ActPos > stParameters.lrPickZPosition + 10.0 THEN
					mcCartesianZMoveAbsolute2.Execute		:= NOT stParameters.bVacuumDeactivate;		
					mcCartesianZMoveAbsolute2.Position		:= stParameters.lrTopZPosition;
					mcCartesianZMoveAbsolute2.Acceleration	:= stParameters.lrPickerAcceleration;
					mcCartesianZMoveAbsolute2.Deceleration	:= stParameters.lrPickerAcceleration;
					mcCartesianZMoveAbsolute2.Velocity		:= stParameters.lrPickerSpeed;
				END_IF
			END_IF

			IF CartesianZAxisRef.NcToPlc.ActPos > stParameters.lrCapCatcherZPosition OR (CartesianZAxisRef.NcToPlc.ActPos > stParameters.lrTopZPosition - 10) THEN
				bCapCatcher1							:= TRUE;
				bCapCatcher2							:= true;
				bCapCatcher3							:= true;
				bCapCatcher4							:= true;
				tonCapCatcher.IN						:= stParameters.bVacuumDeactivate;
			END_IF	
			
			mcCartesianZMoveAbsolute.Execute		:= tonCapCatcher.Q;	
			
			//Dodać sprawdzenie czy gotowy chwytak słomek !!!!!
			//Sprawdzenie pozycji osi pionowej Z i czy wysunięty siłownik chwytaka słomek
			IF ((CartesianZAxisRef.NcToPlc.ActPos > stParameters.lrTopZPosition - 10) OR
				mcCartesianZMoveAbsolute.Done) AND (tonStrawCatcherOut.Q OR NOT stParameters.bStrawCatcherON) THEN
				//Jedź osią poziomą X na pozycję pick
					mcCartesianZMoveAbsolute2.Execute		:= FALSE;
					bCapsBlowON								:= FALSE;
					iSimulationCase							:= 60;
					tonCapCatcher.IN						:= FALSE;
			END_IF
        	
		60:
			bCapCatcher1								:= TRUE;//bCapSucker1;
			bCapCatcher2								:= TRUE;//bCapSucker2;
			bCapCatcher3								:= TRUE;//bCapSucker3;
			bCapCatcher4								:= TRUE;//bCapSucker4;
	
			mcCartesianYMoveAbsolute.Position			:= 3.0;
			mcCartesianYMoveAbsolute.Acceleration		:= stParameters.lrPickerAcceleration;
			mcCartesianYMoveAbsolute.Deceleration		:= stParameters.lrPickerAcceleration;
			mcCartesianYMoveAbsolute.Velocity			:= stParameters.lrPickerSpeed;
			mcCartesianYMoveAbsolute.Execute			:= TRUE;
				
			IF CartesianYAxisRef.NcToPlc.ActPos < 40.0 THEN
				mcCartesianYMoveAbsolute.Execute		:= FALSE;
				iSimulationCase							:= 70;
			END_IF
			
			
			70:
				mcCartesianZMoveAbsolute.Execute			:= TRUE;		
				mcCartesianZMoveAbsolute.Position			:= 360;//stParameters.lrTopZPosition;
				mcCartesianZMoveAbsolute.Acceleration		:= stParameters.lrPickerAcceleration;
				mcCartesianZMoveAbsolute.Deceleration		:= stParameters.lrPickerAcceleration;
				mcCartesianZMoveAbsolute.Velocity			:= stParameters.lrPickerSpeed;
									
					IF mcCartesianZMoveAbsolute.Done THEN
						mcCartesianZMoveAbsolute.Execute	:= FALSE;	
							//Otwórz chwytaki
						bCapCatcher1						:= FALSE;
						bCapCatcher2						:= FALSE;
						bCapCatcher3						:= FALSE;
						bCapCatcher4						:= FALSE;
							//Wyłącz ssawki         		
						bCapSucker[1]						:= FALSE;
						bCapSucker[2]						:= FALSE;
						bCapSucker[3]						:= FALSE;
						bCapSucker[4]						:= FALSE;
						bCapsBlowON							:= TRUE;
						bCapBlow1 							:= TRUE;
						bCapBlow2 							:= TRUE;
						bCapBlow3 							:= TRUE;
						bCapBlow4 							:= TRUE;
						iSimulationCase						:= 80;
					END_IF
				
				80:
					mcCartesianZMoveAbsolute2.Execute		:= TRUE;		
					mcCartesianZMoveAbsolute2.Position		:= stParameters.lrTopZPosition;
					mcCartesianZMoveAbsolute2.Acceleration	:= stParameters.lrPickerAcceleration;
					mcCartesianZMoveAbsolute2.Deceleration	:= stParameters.lrPickerAcceleration;
					mcCartesianZMoveAbsolute2.Velocity		:= stParameters.lrPickerSpeed;
						
						IF 	mcCartesianZMoveAbsolute2.Done THEN
							mcCartesianZMoveAbsolute2.Execute	:= FALSE;
							iSimulationCase						:= 90;
						END_IF
			
				90:
					IF NOT bCapBlow1 AND NOT bCapBlow2 AND NOT bCapBlow3 AND NOT bCapBlow4 THEN
						mcCartesianYMoveAbsolute.Execute		:= TRUE;
						mcCartesianYMoveAbsolute.Position		:= stParameters.lrPickYPosition;
						mcCartesianYMoveAbsolute.Acceleration	:= stParameters.lrPickerAcceleration;
						mcCartesianYMoveAbsolute.Deceleration	:= stParameters.lrPickerAcceleration;
						mcCartesianYMoveAbsolute.Velocity		:= stParameters.lrPickerSpeed;
						iSimulationCase							:= 100;
					END_IF
			
				100:
					IF mcCartesianYMoveAbsolute.Done THEN
						mcCartesianYMoveAbsolute.Execute	:= FALSE;
						iSimulationCase						:= 0;
						bCycleDone							:= TRUE;
						eState								:= E_Station.eDone;
					END_IF

END_CASE
END_ACTION

END_FUNCTION_BLOCK

// ---- POUs/FB/AxisControl/AX8000/FB_AxisAX8000.TcPOU
//==================================================================================================
//							Beckhoff Automation Poland
//									03.01.2023
//
// Code owner: TG
//
// Sample code to handle AX8000 Axis, extends functionality of FB_AxisBase
//
// Used libraries: 
//	Tc2_MC2								|| 3.3.48.0
//	Tc2_System							|| 3.4.26.0
//	Tc2_EtherCAT						|| 3.3.21.0
//
// Used POUs:
//	FB_GetDriveRef
//
// Used DUTs:
//	ST_AxisControlManual
//
//  v1.0	|| TC v 3.1.4024.35		|| First edition
//==================================================================================================
FUNCTION_BLOCK FB_AxisAX8000 EXTENDS FB_AxisBase IMPLEMENTS I_AxisControlPhysical
VAR
	nSafetyState						AT %I*	: BYTE		:= 1;					// 1-ReadyState 0 - SafeState
	nBipolarTorqueLimitValue  			AT %Q*	: UINT		:= 5000; 				// Raw data, linked to Bipolar torque limit value
	_bWritingEncoderOffset						: BOOL;								// Forces MC_Power disable when encoder offset is written

	// Properties
	{attribute 'hide'}
	_bHoldingBrakePresent						: BOOL;
	{attribute 'hide'}
	_bHoldingBrakeLocked						: BOOL;
	{attribute 'hide'}
	_bHoldingBrakeUnlocked						: BOOL;
	{attribute 'hide'}
	_stDriveAddress								: Tc2_MC2.ST_DriveAddress;
	{attribute 'hide'}
	_stDriveRef									: Tc2_EtherCAT.ST_DriveRef;
	// FBs
	{attribute 'hide'}
	fbSetPositionOffset							: Tc2_MC2_Drive.FB_CoEAX8000SetPositionOffset;
	{attribute 'hide'}
	_stSetPosOffs 								: Tc2_MC2.ST_McOutputs;
	{attribute 'hide'}
	fbDeletePositionOffset						: Tc2_MC2_Drive.FB_CoEAX8000DeletePositionOffset;
	{attribute 'hide'}
	_stDeletePosOffs 							: Tc2_MC2.ST_McOutputs;
END_VAR

SUPER^();

{attribute 'monitoring' := 'variable'}
PROPERTY bHoldingBrakeLocked 					: BOOL
GET
bHoldingBrakeLocked								:= _bHoldingBrakeLocked;
END_GET
SET
_bHoldingBrakeLocked							:= bHoldingBrakeLocked;
END_SET
END_PROPERTY

{attribute 'monitoring' := 'variable'}
PROPERTY bHoldingBrakePresent 					: BOOL
GET
bHoldingBrakePresent								:= _bHoldingBrakePresent;
END_GET
SET
_bHoldingBrakePresent							:= bHoldingBrakePresent;
END_SET
END_PROPERTY

{attribute 'monitoring' := 'variable'}
PROPERTY bHoldingBrakeUnlocked 					: BOOL
GET
bHoldingBrakeUnlocked							:= _bHoldingBrakeUnlocked;
END_GET
SET
_bHoldingBrakeUnlocked							:= bHoldingBrakeUnlocked;
END_SET
END_PROPERTY

METHOD BrakeControl 							: REFERENCE TO Tc2_MC2.ST_McOutputs
VAR_INPUT
	bForceLock 									: BOOL;								// 
	bForceUnlock								: BOOL;								// 
END_VAR
VAR_INST
	{attribute 'hide'}
	fbBrakeCtrl									: FB_HoldingBrakeCtrlAX8000;
	{attribute 'hide'}
	ftBusy										: F_TRIG;
END_VAR
VAR
	{attribute 'hide'}
	Out											: Tc2_MC2.ST_McOutputs;
END_VAR
fbBrakeCtrl(		bForceLock				:= bForceLock, 
					bForceUnlock			:= bForceUnlock, 
					stDriveRef				:= _stDriveRef, 
					bBusy					=> Out.Busy, 
					bError					=> Out.Error);

IF Out.Error THEN
	Out.ErrorID								:= fbBrakeCtrl.iAdsErrId + fbBrakeCtrl.iCANopenErrId;
END_IF
					
ftBusy(CLK:= Out.Busy, Q=> );
IF ftBusy.Q THEN
	Out.Done								:= NOT Out.Error;
END_IF

BrakeControl								REF= Out;
END_METHOD

METHOD BrakeForceLock 							: REFERENCE TO Tc2_MC2.ST_McOutputs
BrakeForceLock REF= BrakeControl(bForceLock := TRUE, bForceUnlock := FALSE);
END_METHOD

METHOD BrakeForceUnlock 						: REFERENCE TO Tc2_MC2.ST_McOutputs
BrakeForceUnlock REF= BrakeControl(bForceLock := FALSE, bForceUnlock := TRUE);
END_METHOD

METHOD BrakePresent 							: REFERENCE TO Tc2_MC2.ST_McOutputs
VAR_INPUT
	bExecute									: BOOL;
END_VAR
VAR_INST
	{attribute 'hide'}
	fbRead										: Tc2_EtherCAT.FB_CoERead_ByDriveRef;
	{attribute 'hide'}
	ftRead										: F_TRIG;
	{attribute 'hide'}
	nData										: WORD;
END_VAR
VAR
	Out											: Tc2_MC2.ST_McOutputs;
END_VAR
fbRead			(	stDriveRef				:= _stDriveRef, 
					nIndex					:= 16#3000 + (_stDriveRef.nDriveNo * 16#400), 
					nSubIndex				:= 16#01, 
					pDstBuf					:= ADR(nData), 
					cbBufLen				:= SIZEOF(nData), 
					bExecute				:= bExecute,
					bBusy					=> Out.Busy, 
					bError					=> Out.Error, 
					iAdsErrId				=> , 
					iCANopenErrId			=> );

IF Out.Error THEN
	Out.ErrorID								:= fbRead.iAdsErrId + fbRead.iCANopenErrId;
END_IF
					
ftRead(CLK:= Out.Busy, Q=> );
IF ftRead.Q THEN
	Out.Done								:= NOT Out.Error;
	bHoldingBrakePresent						:= nData.0;
END_IF

BrakePresent								REF= Out;
END_METHOD

METHOD BrakeReleaseForce 						: REFERENCE TO Tc2_MC2.ST_McOutputs
BrakeReleaseForce REF= BrakeControl(bForceLock := FALSE, bForceUnlock := FALSE);
END_METHOD

